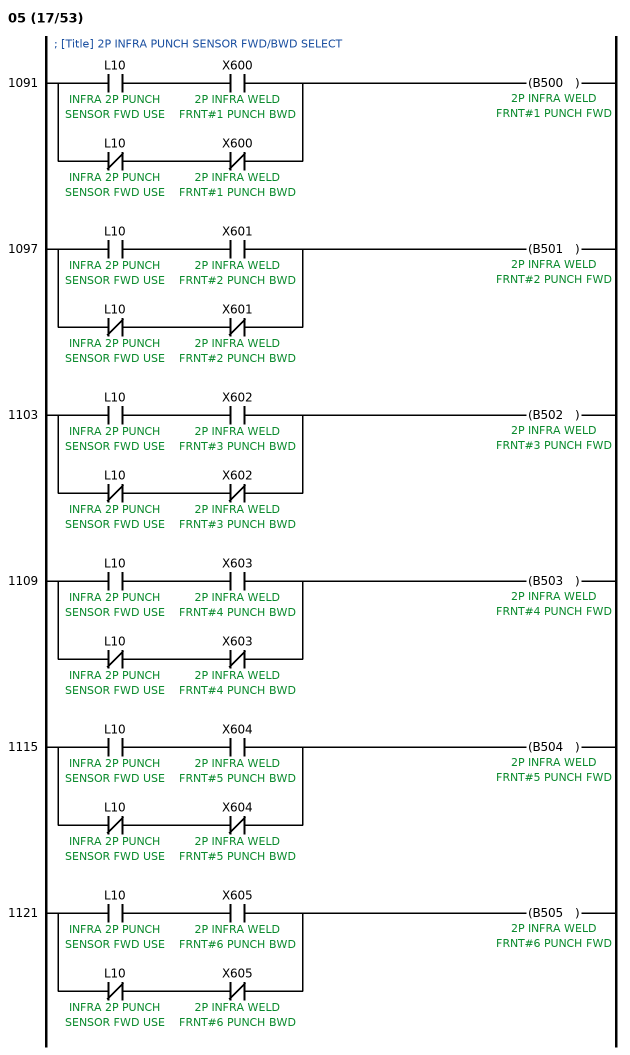
; [Title] 2P INFRA PUNCH SENSOR FWD/BWD SELECT
1091  LD      L10  ; INFRA 2P PUNCH SENSOR FWD USE
      AND     X600  ; 2P INFRA WELD FRNT#1 PUNCH BWD
      LDI     L10  ; INFRA 2P PUNCH SENSOR FWD USE
      ANI     X600  ; 2P INFRA WELD FRNT#1 PUNCH BWD
      ORB
      OUT     B500  ; 2P INFRA WELD FRNT#1 PUNCH FWD
1097  LD      L10  ; INFRA 2P PUNCH SENSOR FWD USE
      AND     X601  ; 2P INFRA WELD FRNT#2 PUNCH BWD
      LDI     L10  ; INFRA 2P PUNCH SENSOR FWD USE
      ANI     X601  ; 2P INFRA WELD FRNT#2 PUNCH BWD
      ORB
      OUT     B501  ; 2P INFRA WELD FRNT#2 PUNCH FWD
1103  LD      L10  ; INFRA 2P PUNCH SENSOR FWD USE
      AND     X602  ; 2P INFRA WELD FRNT#3 PUNCH BWD
      LDI     L10  ; INFRA 2P PUNCH SENSOR FWD USE
      ANI     X602  ; 2P INFRA WELD FRNT#3 PUNCH BWD
      ORB
      OUT     B502  ; 2P INFRA WELD FRNT#3 PUNCH FWD
1109  LD      L10  ; INFRA 2P PUNCH SENSOR FWD USE
      AND     X603  ; 2P INFRA WELD FRNT#4 PUNCH BWD
      LDI     L10  ; INFRA 2P PUNCH SENSOR FWD USE
      ANI     X603  ; 2P INFRA WELD FRNT#4 PUNCH BWD
      ORB
      OUT     B503  ; 2P INFRA WELD FRNT#4 PUNCH FWD
1115  LD      L10  ; INFRA 2P PUNCH SENSOR FWD USE
      AND     X604  ; 2P INFRA WELD FRNT#5 PUNCH BWD
      LDI     L10  ; INFRA 2P PUNCH SENSOR FWD USE
      ANI     X604  ; 2P INFRA WELD FRNT#5 PUNCH BWD
      ORB
      OUT     B504  ; 2P INFRA WELD FRNT#5 PUNCH FWD
1121  LD      L10  ; INFRA 2P PUNCH SENSOR FWD USE
      AND     X605  ; 2P INFRA WELD FRNT#6 PUNCH BWD
      LDI     L10  ; INFRA 2P PUNCH SENSOR FWD USE
      ANI     X605  ; 2P INFRA WELD FRNT#6 PUNCH BWD
      ORB
      OUT     B505  ; 2P INFRA WELD FRNT#6 PUNCH FWD
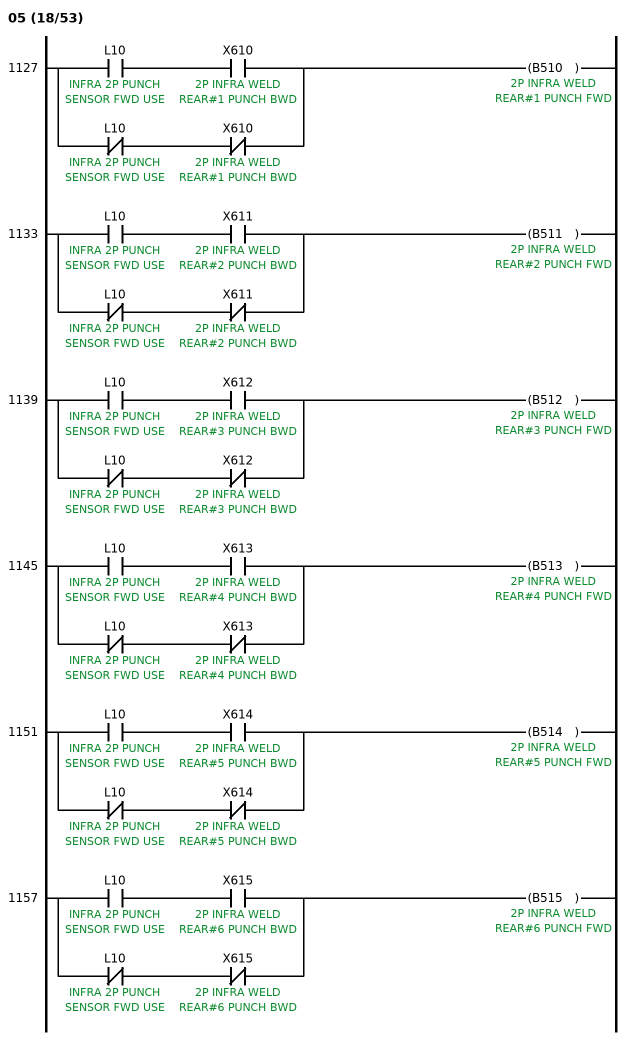
1127  LD      L10  ; INFRA 2P PUNCH SENSOR FWD USE
      AND     X610  ; 2P INFRA WELD REAR#1 PUNCH BWD
      LDI     L10  ; INFRA 2P PUNCH SENSOR FWD USE
      ANI     X610  ; 2P INFRA WELD REAR#1 PUNCH BWD
      ORB
      OUT     B510  ; 2P INFRA WELD REAR#1 PUNCH FWD
1133  LD      L10  ; INFRA 2P PUNCH SENSOR FWD USE
      AND     X611  ; 2P INFRA WELD REAR#2 PUNCH BWD
      LDI     L10  ; INFRA 2P PUNCH SENSOR FWD USE
      ANI     X611  ; 2P INFRA WELD REAR#2 PUNCH BWD
      ORB
      OUT     B511  ; 2P INFRA WELD REAR#2 PUNCH FWD
1139  LD      L10  ; INFRA 2P PUNCH SENSOR FWD USE
      AND     X612  ; 2P INFRA WELD REAR#3 PUNCH BWD
      LDI     L10  ; INFRA 2P PUNCH SENSOR FWD USE
      ANI     X612  ; 2P INFRA WELD REAR#3 PUNCH BWD
      ORB
      OUT     B512  ; 2P INFRA WELD REAR#3 PUNCH FWD
1145  LD      L10  ; INFRA 2P PUNCH SENSOR FWD USE
      AND     X613  ; 2P INFRA WELD REAR#4 PUNCH BWD
      LDI     L10  ; INFRA 2P PUNCH SENSOR FWD USE
      ANI     X613  ; 2P INFRA WELD REAR#4 PUNCH BWD
      ORB
      OUT     B513  ; 2P INFRA WELD REAR#4 PUNCH FWD
1151  LD      L10  ; INFRA 2P PUNCH SENSOR FWD USE
      AND     X614  ; 2P INFRA WELD REAR#5 PUNCH BWD
      LDI     L10  ; INFRA 2P PUNCH SENSOR FWD USE
      ANI     X614  ; 2P INFRA WELD REAR#5 PUNCH BWD
      ORB
      OUT     B514  ; 2P INFRA WELD REAR#5 PUNCH FWD
1157  LD      L10  ; INFRA 2P PUNCH SENSOR FWD USE
      AND     X615  ; 2P INFRA WELD REAR#6 PUNCH BWD
      LDI     L10  ; INFRA 2P PUNCH SENSOR FWD USE
      ANI     X615  ; 2P INFRA WELD REAR#6 PUNCH BWD
      ORB
      OUT     B515  ; 2P INFRA WELD REAR#6 PUNCH FWD
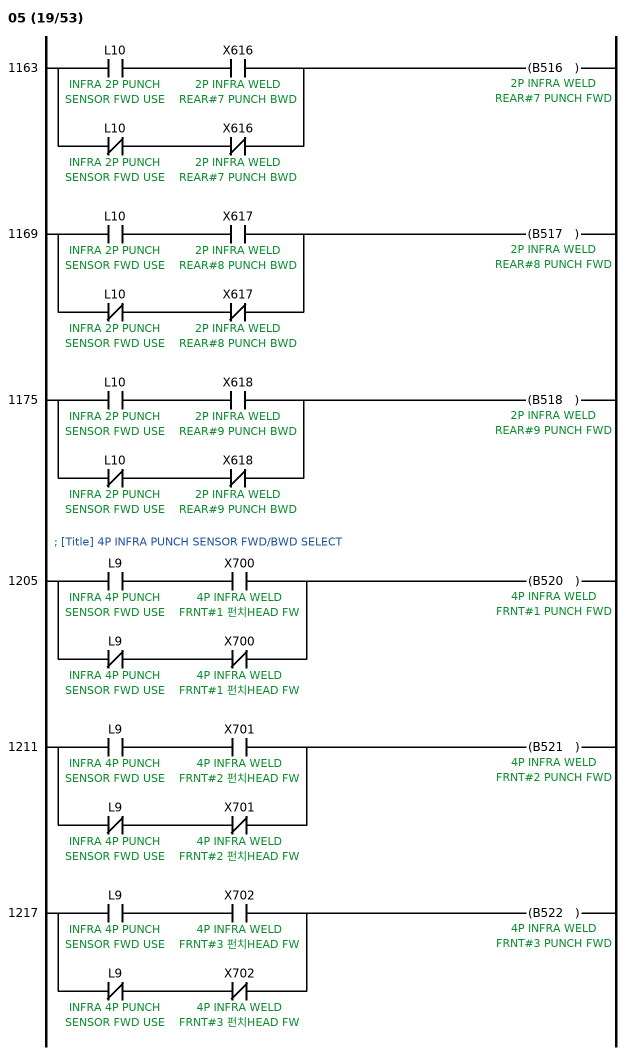
1163  LD      L10  ; INFRA 2P PUNCH SENSOR FWD USE
      AND     X616  ; 2P INFRA WELD REAR#7 PUNCH BWD
      LDI     L10  ; INFRA 2P PUNCH SENSOR FWD USE
      ANI     X616  ; 2P INFRA WELD REAR#7 PUNCH BWD
      ORB
      OUT     B516  ; 2P INFRA WELD REAR#7 PUNCH FWD
1169  LD      L10  ; INFRA 2P PUNCH SENSOR FWD USE
      AND     X617  ; 2P INFRA WELD REAR#8 PUNCH BWD
      LDI     L10  ; INFRA 2P PUNCH SENSOR FWD USE
      ANI     X617  ; 2P INFRA WELD REAR#8 PUNCH BWD
      ORB
      OUT     B517  ; 2P INFRA WELD REAR#8 PUNCH FWD
1175  LD      L10  ; INFRA 2P PUNCH SENSOR FWD USE
      AND     X618  ; 2P INFRA WELD REAR#9 PUNCH BWD
      LDI     L10  ; INFRA 2P PUNCH SENSOR FWD USE
      ANI     X618  ; 2P INFRA WELD REAR#9 PUNCH BWD
      ORB
      OUT     B518  ; 2P INFRA WELD REAR#9 PUNCH FWD
; [Title] 4P INFRA PUNCH SENSOR FWD/BWD SELECT
1205  LD      L9  ; INFRA 4P PUNCH SENSOR FWD USE
      AND     X700  ; 4P INFRA WELD FRNT#1 펀치HEAD FW
      LDI     L9  ; INFRA 4P PUNCH SENSOR FWD USE
      ANI     X700  ; 4P INFRA WELD FRNT#1 펀치HEAD FW
      ORB
      OUT     B520  ; 4P INFRA WELD FRNT#1 PUNCH FWD
1211  LD      L9  ; INFRA 4P PUNCH SENSOR FWD USE
      AND     X701  ; 4P INFRA WELD FRNT#2 펀치HEAD FW
      LDI     L9  ; INFRA 4P PUNCH SENSOR FWD USE
      ANI     X701  ; 4P INFRA WELD FRNT#2 펀치HEAD FW
      ORB
      OUT     B521  ; 4P INFRA WELD FRNT#2 PUNCH FWD
1217  LD      L9  ; INFRA 4P PUNCH SENSOR FWD USE
      AND     X702  ; 4P INFRA WELD FRNT#3 펀치HEAD FW
      LDI     L9  ; INFRA 4P PUNCH SENSOR FWD USE
      ANI     X702  ; 4P INFRA WELD FRNT#3 펀치HEAD FW
      ORB
      OUT     B522  ; 4P INFRA WELD FRNT#3 PUNCH FWD
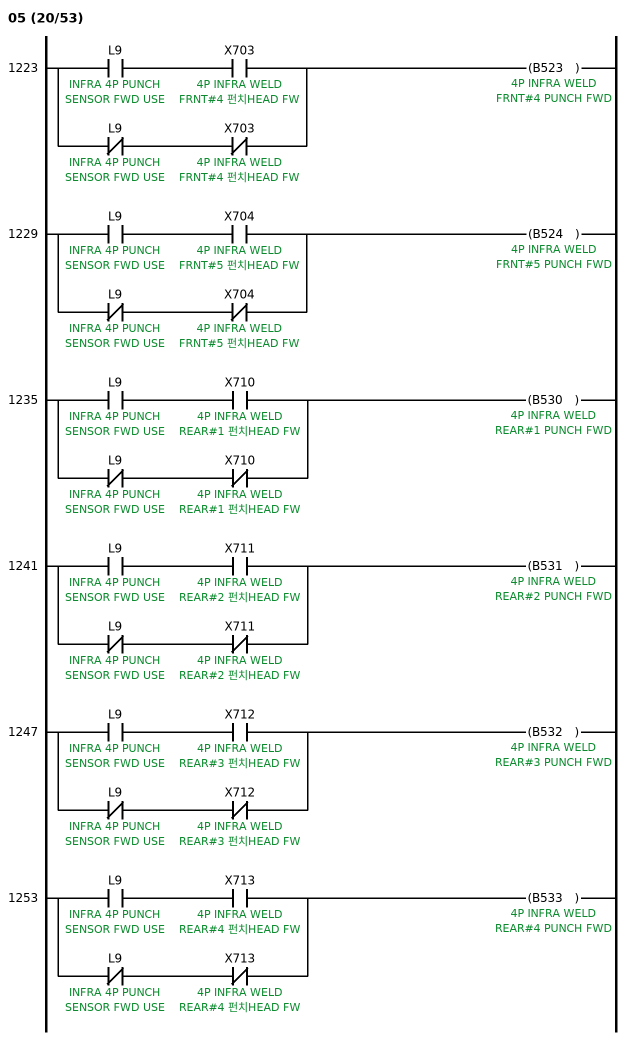
1223  LD      L9  ; INFRA 4P PUNCH SENSOR FWD USE
      AND     X703  ; 4P INFRA WELD FRNT#4 펀치HEAD FW
      LDI     L9  ; INFRA 4P PUNCH SENSOR FWD USE
      ANI     X703  ; 4P INFRA WELD FRNT#4 펀치HEAD FW
      ORB
      OUT     B523  ; 4P INFRA WELD FRNT#4 PUNCH FWD
1229  LD      L9  ; INFRA 4P PUNCH SENSOR FWD USE
      AND     X704  ; 4P INFRA WELD FRNT#5 펀치HEAD FW
      LDI     L9  ; INFRA 4P PUNCH SENSOR FWD USE
      ANI     X704  ; 4P INFRA WELD FRNT#5 펀치HEAD FW
      ORB
      OUT     B524  ; 4P INFRA WELD FRNT#5 PUNCH FWD
1235  LD      L9  ; INFRA 4P PUNCH SENSOR FWD USE
      AND     X710  ; 4P INFRA WELD REAR#1 펀치HEAD FW
      LDI     L9  ; INFRA 4P PUNCH SENSOR FWD USE
      ANI     X710  ; 4P INFRA WELD REAR#1 펀치HEAD FW
      ORB
      OUT     B530  ; 4P INFRA WELD REAR#1 PUNCH FWD
1241  LD      L9  ; INFRA 4P PUNCH SENSOR FWD USE
      AND     X711  ; 4P INFRA WELD REAR#2 펀치HEAD FW
      LDI     L9  ; INFRA 4P PUNCH SENSOR FWD USE
      ANI     X711  ; 4P INFRA WELD REAR#2 펀치HEAD FW
      ORB
      OUT     B531  ; 4P INFRA WELD REAR#2 PUNCH FWD
1247  LD      L9  ; INFRA 4P PUNCH SENSOR FWD USE
      AND     X712  ; 4P INFRA WELD REAR#3 펀치HEAD FW
      LDI     L9  ; INFRA 4P PUNCH SENSOR FWD USE
      ANI     X712  ; 4P INFRA WELD REAR#3 펀치HEAD FW
      ORB
      OUT     B532  ; 4P INFRA WELD REAR#3 PUNCH FWD
1253  LD      L9  ; INFRA 4P PUNCH SENSOR FWD USE
      AND     X713  ; 4P INFRA WELD REAR#4 펀치HEAD FW
      LDI     L9  ; INFRA 4P PUNCH SENSOR FWD USE
      ANI     X713  ; 4P INFRA WELD REAR#4 펀치HEAD FW
      ORB
      OUT     B533  ; 4P INFRA WELD REAR#4 PUNCH FWD
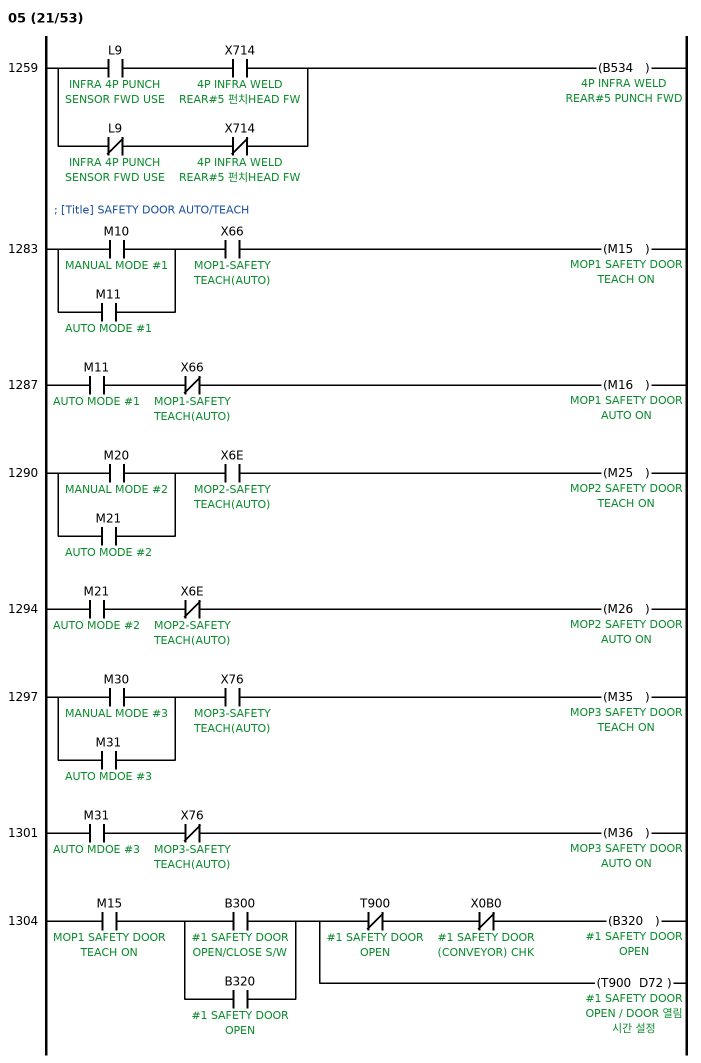
1259  LD      L9  ; INFRA 4P PUNCH SENSOR FWD USE
      AND     X714  ; 4P INFRA WELD REAR#5 펀치HEAD FW
      LDI     L9  ; INFRA 4P PUNCH SENSOR FWD USE
      ANI     X714  ; 4P INFRA WELD REAR#5 펀치HEAD FW
      ORB
      OUT     B534  ; 4P INFRA WELD REAR#5 PUNCH FWD
; [Title] SAFETY DOOR AUTO/TEACH
1283  LD      M10  ; MANUAL MODE #1
      OR      M11  ; AUTO MODE #1
      AND     X66  ; MOP1-SAFETY TEACH(AUTO)
      OUT     M15  ; MOP1 SAFETY DOOR TEACH ON
1287  LD      M11  ; AUTO MODE #1
      ANI     X66  ; MOP1-SAFETY TEACH(AUTO)
      OUT     M16  ; MOP1 SAFETY DOOR AUTO ON
1290  LD      M20  ; MANUAL MODE #2
      OR      M21  ; AUTO MODE #2
      AND     X6E  ; MOP2-SAFETY TEACH(AUTO)
      OUT     M25  ; MOP2 SAFETY DOOR TEACH ON
1294  LD      M21  ; AUTO MODE #2
      ANI     X6E  ; MOP2-SAFETY TEACH(AUTO)
      OUT     M26  ; MOP2 SAFETY DOOR AUTO ON
1297  LD      M30  ; MANUAL MODE #3
      OR      M31  ; AUTO MDOE #3
      AND     X76  ; MOP3-SAFETY TEACH(AUTO)
      OUT     M35  ; MOP3 SAFETY DOOR TEACH ON
1301  LD      M31  ; AUTO MDOE #3
      ANI     X76  ; MOP3-SAFETY TEACH(AUTO)
      OUT     M36  ; MOP3 SAFETY DOOR AUTO ON
1304  LD      M15  ; MOP1 SAFETY DOOR TEACH ON
      LD      B300  ; #1 SAFETY DOOR  OPEN/CLOSE S/W
      OR      B320  ; #1 SAFETY DOOR  OPEN
      ANB
      MPS
      ANI     T900  ; #1 SAFETY DOOR  OPEN
      ANI     X0B0  ; #1 SAFETY DOOR (CONVEYOR) CHK
      OUT     B320  ; #1 SAFETY DOOR  OPEN
      MPP
      OUT     T900 D72  ; #1 SAFETY DOOR  OPEN / DOOR 열림 시간 설정
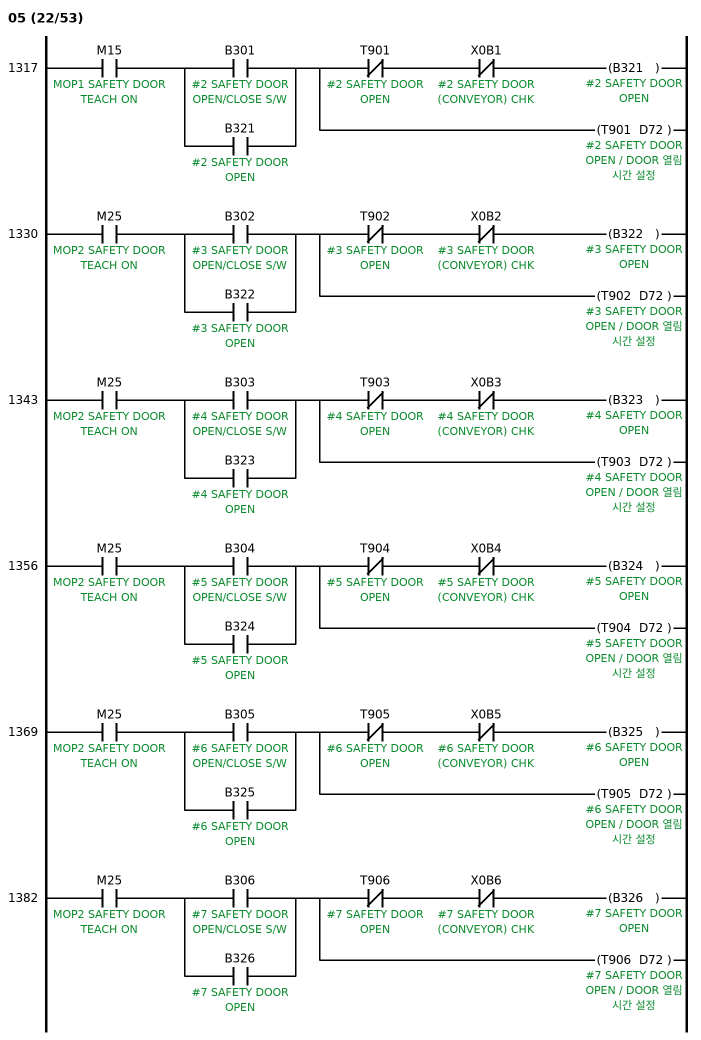
1317  LD      M15  ; MOP1 SAFETY DOOR TEACH ON
      LD      B301  ; #2 SAFETY DOOR  OPEN/CLOSE S/W
      OR      B321  ; #2 SAFETY DOOR  OPEN
      ANB
      MPS
      ANI     T901  ; #2 SAFETY DOOR  OPEN
      ANI     X0B1  ; #2 SAFETY DOOR (CONVEYOR) CHK
      OUT     B321  ; #2 SAFETY DOOR  OPEN
      MPP
      OUT     T901 D72  ; #2 SAFETY DOOR  OPEN / DOOR 열림 시간 설정
1330  LD      M25  ; MOP2 SAFETY DOOR TEACH ON
      LD      B302  ; #3 SAFETY DOOR  OPEN/CLOSE S/W
      OR      B322  ; #3 SAFETY DOOR  OPEN
      ANB
      MPS
      ANI     T902  ; #3 SAFETY DOOR  OPEN
      ANI     X0B2  ; #3 SAFETY DOOR (CONVEYOR) CHK
      OUT     B322  ; #3 SAFETY DOOR  OPEN
      MPP
      OUT     T902 D72  ; #3 SAFETY DOOR  OPEN / DOOR 열림 시간 설정
1343  LD      M25  ; MOP2 SAFETY DOOR TEACH ON
      LD      B303  ; #4 SAFETY DOOR  OPEN/CLOSE S/W
      OR      B323  ; #4 SAFETY DOOR  OPEN
      ANB
      MPS
      ANI     T903  ; #4 SAFETY DOOR  OPEN
      ANI     X0B3  ; #4 SAFETY DOOR (CONVEYOR) CHK
      OUT     B323  ; #4 SAFETY DOOR  OPEN
      MPP
      OUT     T903 D72  ; #4 SAFETY DOOR  OPEN / DOOR 열림 시간 설정
1356  LD      M25  ; MOP2 SAFETY DOOR TEACH ON
      LD      B304  ; #5 SAFETY DOOR  OPEN/CLOSE S/W
      OR      B324  ; #5 SAFETY DOOR  OPEN
      ANB
      MPS
      ANI     T904  ; #5 SAFETY DOOR  OPEN
      ANI     X0B4  ; #5 SAFETY DOOR (CONVEYOR) CHK
      OUT     B324  ; #5 SAFETY DOOR  OPEN
      MPP
      OUT     T904 D72  ; #5 SAFETY DOOR  OPEN / DOOR 열림 시간 설정
1369  LD      M25  ; MOP2 SAFETY DOOR TEACH ON
      LD      B305  ; #6 SAFETY DOOR  OPEN/CLOSE S/W
      OR      B325  ; #6 SAFETY DOOR  OPEN
      ANB
      MPS
      ANI     T905  ; #6 SAFETY DOOR  OPEN
      ANI     X0B5  ; #6 SAFETY DOOR (CONVEYOR) CHK
      OUT     B325  ; #6 SAFETY DOOR  OPEN
      MPP
      OUT     T905 D72  ; #6 SAFETY DOOR  OPEN / DOOR 열림 시간 설정
1382  LD      M25  ; MOP2 SAFETY DOOR TEACH ON
      LD      B306  ; #7 SAFETY DOOR  OPEN/CLOSE S/W
      OR      B326  ; #7 SAFETY DOOR  OPEN
      ANB
      MPS
      ANI     T906  ; #7 SAFETY DOOR  OPEN
      ANI     X0B6  ; #7 SAFETY DOOR (CONVEYOR) CHK
      OUT     B326  ; #7 SAFETY DOOR  OPEN
      MPP
      OUT     T906 D72  ; #7 SAFETY DOOR  OPEN / DOOR 열림 시간 설정
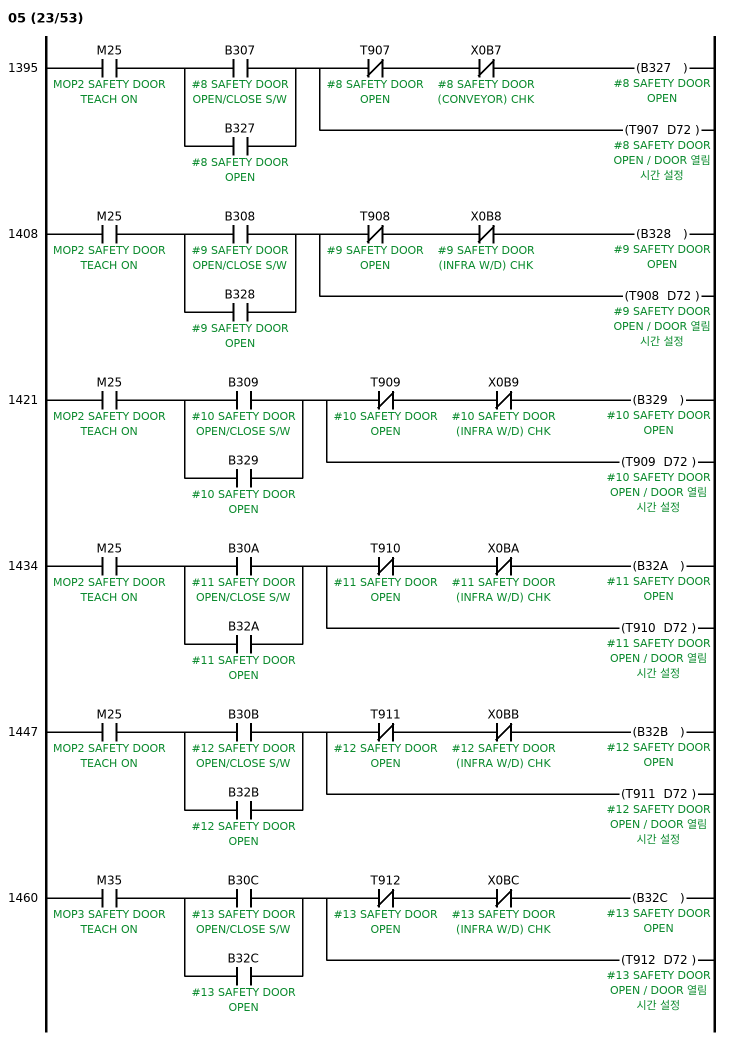
1395  LD      M25  ; MOP2 SAFETY DOOR TEACH ON
      LD      B307  ; #8 SAFETY DOOR  OPEN/CLOSE S/W
      OR      B327  ; #8 SAFETY DOOR  OPEN
      ANB
      MPS
      ANI     T907  ; #8 SAFETY DOOR  OPEN
      ANI     X0B7  ; #8 SAFETY DOOR (CONVEYOR) CHK
      OUT     B327  ; #8 SAFETY DOOR  OPEN
      MPP
      OUT     T907 D72  ; #8 SAFETY DOOR  OPEN / DOOR 열림 시간 설정
1408  LD      M25  ; MOP2 SAFETY DOOR TEACH ON
      LD      B308  ; #9 SAFETY DOOR  OPEN/CLOSE S/W
      OR      B328  ; #9 SAFETY DOOR  OPEN
      ANB
      MPS
      ANI     T908  ; #9 SAFETY DOOR  OPEN
      ANI     X0B8  ; #9 SAFETY DOOR (INFRA W/D) CHK
      OUT     B328  ; #9 SAFETY DOOR  OPEN
      MPP
      OUT     T908 D72  ; #9 SAFETY DOOR  OPEN / DOOR 열림 시간 설정
1421  LD      M25  ; MOP2 SAFETY DOOR TEACH ON
      LD      B309  ; #10 SAFETY DOOR OPEN/CLOSE S/W
      OR      B329  ; #10 SAFETY DOOR OPEN
      ANB
      MPS
      ANI     T909  ; #10 SAFETY DOOR OPEN
      ANI     X0B9  ; #10 SAFETY DOOR (INFRA W/D) CHK
      OUT     B329  ; #10 SAFETY DOOR OPEN
      MPP
      OUT     T909 D72  ; #10 SAFETY DOOR OPEN / DOOR 열림 시간 설정
1434  LD      M25  ; MOP2 SAFETY DOOR TEACH ON
      LD      B30A  ; #11 SAFETY DOOR OPEN/CLOSE S/W
      OR      B32A  ; #11 SAFETY DOOR OPEN
      ANB
      MPS
      ANI     T910  ; #11 SAFETY DOOR OPEN
      ANI     X0BA  ; #11 SAFETY DOOR (INFRA W/D) CHK
      OUT     B32A  ; #11 SAFETY DOOR OPEN
      MPP
      OUT     T910 D72  ; #11 SAFETY DOOR OPEN / DOOR 열림 시간 설정
1447  LD      M25  ; MOP2 SAFETY DOOR TEACH ON
      LD      B30B  ; #12 SAFETY DOOR OPEN/CLOSE S/W
      OR      B32B  ; #12 SAFETY DOOR OPEN
      ANB
      MPS
      ANI     T911  ; #12 SAFETY DOOR OPEN
      ANI     X0BB  ; #12 SAFETY DOOR (INFRA W/D) CHK
      OUT     B32B  ; #12 SAFETY DOOR OPEN
      MPP
      OUT     T911 D72  ; #12 SAFETY DOOR OPEN / DOOR 열림 시간 설정
1460  LD      M35  ; MOP3 SAFETY DOOR TEACH ON
      LD      B30C  ; #13 SAFETY DOOR OPEN/CLOSE S/W
      OR      B32C  ; #13 SAFETY DOOR OPEN
      ANB
      MPS
      ANI     T912  ; #13 SAFETY DOOR OPEN
      ANI     X0BC  ; #13 SAFETY DOOR (INFRA W/D) CHK
      OUT     B32C  ; #13 SAFETY DOOR OPEN
      MPP
      OUT     T912 D72  ; #13 SAFETY DOOR OPEN / DOOR 열림 시간 설정
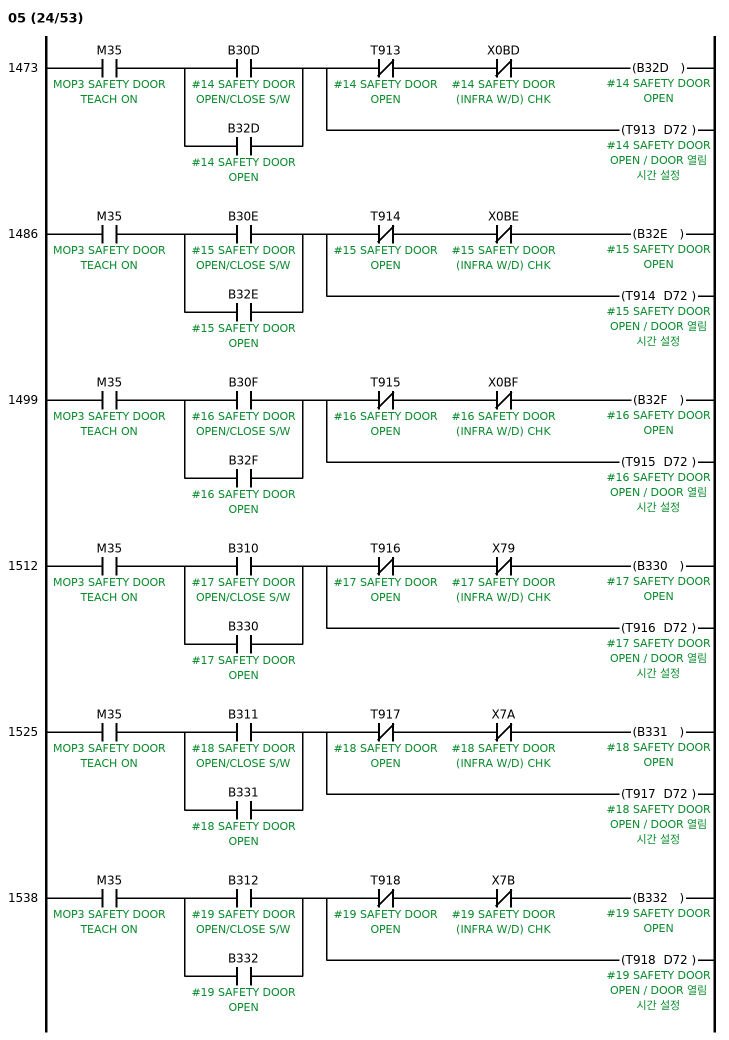
1473  LD      M35  ; MOP3 SAFETY DOOR TEACH ON
      LD      B30D  ; #14 SAFETY DOOR OPEN/CLOSE S/W
      OR      B32D  ; #14 SAFETY DOOR OPEN
      ANB
      MPS
      ANI     T913  ; #14 SAFETY DOOR OPEN
      ANI     X0BD  ; #14 SAFETY DOOR (INFRA W/D) CHK
      OUT     B32D  ; #14 SAFETY DOOR OPEN
      MPP
      OUT     T913 D72  ; #14 SAFETY DOOR OPEN / DOOR 열림 시간 설정
1486  LD      M35  ; MOP3 SAFETY DOOR TEACH ON
      LD      B30E  ; #15 SAFETY DOOR OPEN/CLOSE S/W
      OR      B32E  ; #15 SAFETY DOOR OPEN
      ANB
      MPS
      ANI     T914  ; #15 SAFETY DOOR OPEN
      ANI     X0BE  ; #15 SAFETY DOOR (INFRA W/D) CHK
      OUT     B32E  ; #15 SAFETY DOOR OPEN
      MPP
      OUT     T914 D72  ; #15 SAFETY DOOR OPEN / DOOR 열림 시간 설정
1499  LD      M35  ; MOP3 SAFETY DOOR TEACH ON
      LD      B30F  ; #16 SAFETY DOOR OPEN/CLOSE S/W
      OR      B32F  ; #16 SAFETY DOOR OPEN
      ANB
      MPS
      ANI     T915  ; #16 SAFETY DOOR OPEN
      ANI     X0BF  ; #16 SAFETY DOOR (INFRA W/D) CHK
      OUT     B32F  ; #16 SAFETY DOOR OPEN
      MPP
      OUT     T915 D72  ; #16 SAFETY DOOR OPEN / DOOR 열림 시간 설정
1512  LD      M35  ; MOP3 SAFETY DOOR TEACH ON
      LD      B310  ; #17 SAFETY DOOR OPEN/CLOSE S/W
      OR      B330  ; #17 SAFETY DOOR OPEN
      ANB
      MPS
      ANI     T916  ; #17 SAFETY DOOR OPEN
      ANI     X79  ; #17 SAFETY DOOR (INFRA W/D) CHK
      OUT     B330  ; #17 SAFETY DOOR OPEN
      MPP
      OUT     T916 D72  ; #17 SAFETY DOOR OPEN / DOOR 열림 시간 설정
1525  LD      M35  ; MOP3 SAFETY DOOR TEACH ON
      LD      B311  ; #18 SAFETY DOOR OPEN/CLOSE S/W
      OR      B331  ; #18 SAFETY DOOR OPEN
      ANB
      MPS
      ANI     T917  ; #18 SAFETY DOOR OPEN
      ANI     X7A  ; #18 SAFETY DOOR (INFRA W/D) CHK
      OUT     B331  ; #18 SAFETY DOOR OPEN
      MPP
      OUT     T917 D72  ; #18 SAFETY DOOR OPEN / DOOR 열림 시간 설정
1538  LD      M35  ; MOP3 SAFETY DOOR TEACH ON
      LD      B312  ; #19 SAFETY DOOR OPEN/CLOSE S/W
      OR      B332  ; #19 SAFETY DOOR OPEN
      ANB
      MPS
      ANI     T918  ; #19 SAFETY DOOR OPEN
      ANI     X7B  ; #19 SAFETY DOOR (INFRA W/D) CHK
      OUT     B332  ; #19 SAFETY DOOR OPEN
      MPP
      OUT     T918 D72  ; #19 SAFETY DOOR OPEN / DOOR 열림 시간 설정
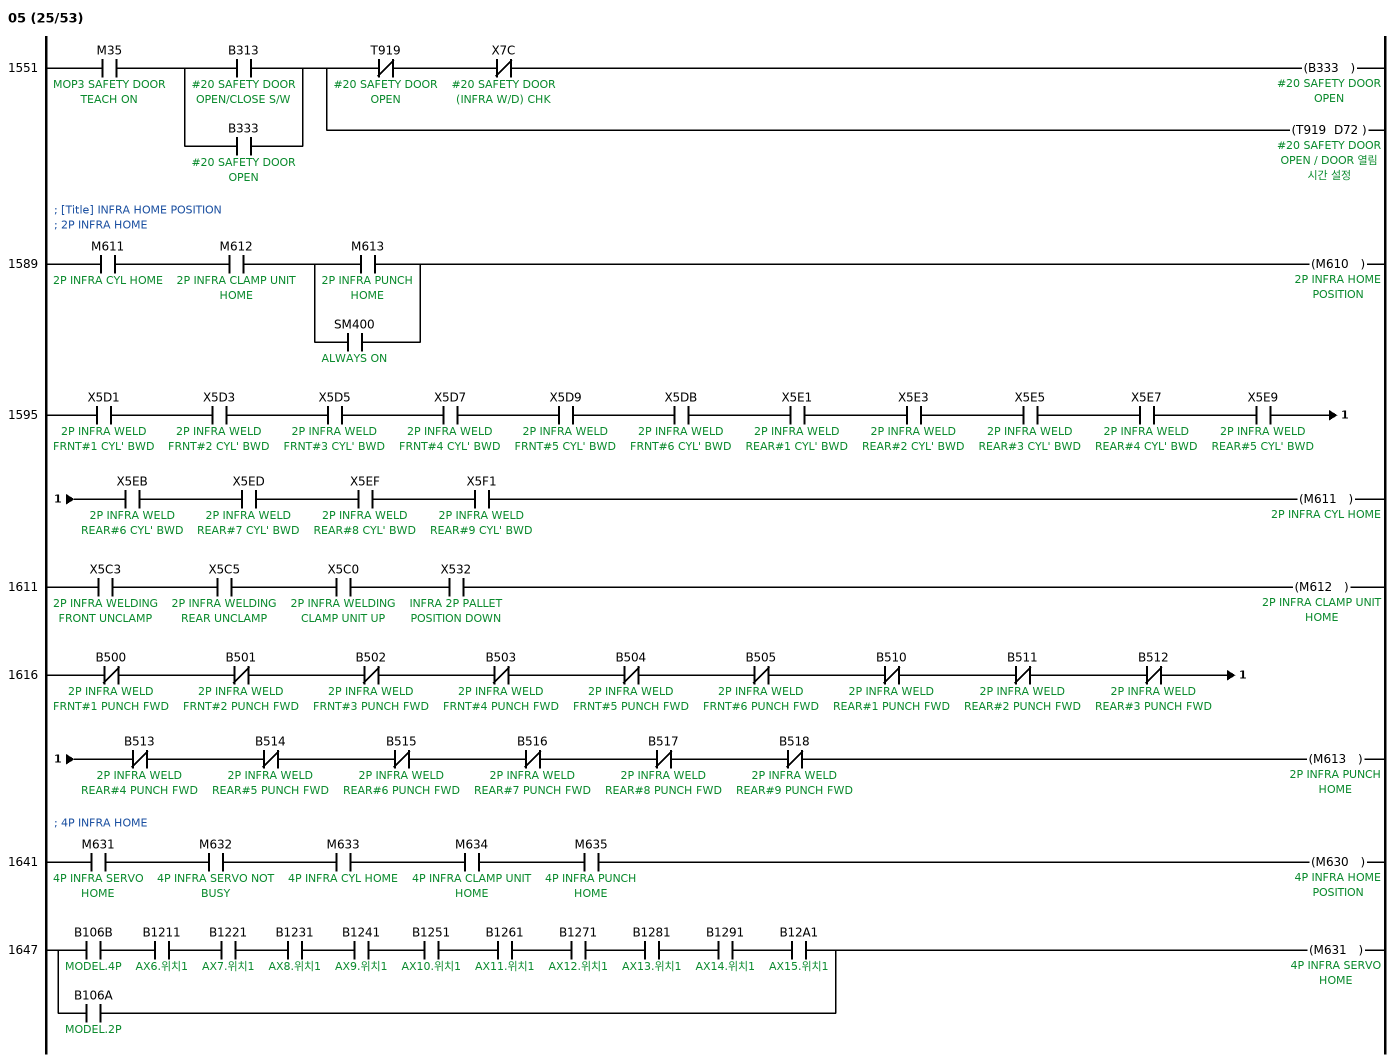
1551  LD      M35  ; MOP3 SAFETY DOOR TEACH ON
      LD      B313  ; #20 SAFETY DOOR OPEN/CLOSE S/W
      OR      B333  ; #20 SAFETY DOOR OPEN
      ANB
      MPS
      ANI     T919  ; #20 SAFETY DOOR OPEN
      ANI     X7C  ; #20 SAFETY DOOR (INFRA W/D) CHK
      OUT     B333  ; #20 SAFETY DOOR OPEN
      MPP
      OUT     T919 D72  ; #20 SAFETY DOOR OPEN / DOOR 열림 시간 설정
; [Title] INFRA HOME POSITION
; 2P INFRA HOME
1589  LD      M611  ; 2P INFRA CYL HOME
      AND     M612  ; 2P INFRA CLAMP UNIT HOME
      LD      M613  ; 2P INFRA PUNCH HOME
      OR      SM400  ; ALWAYS ON
      ANB
      OUT     M610  ; 2P INFRA HOME POSITION
1595  LD      X5D1  ; 2P INFRA WELD FRNT#1 CYL' BWD
      AND     X5D3  ; 2P INFRA WELD FRNT#2 CYL' BWD
      AND     X5D5  ; 2P INFRA WELD FRNT#3 CYL' BWD
      AND     X5D7  ; 2P INFRA WELD FRNT#4 CYL' BWD
      AND     X5D9  ; 2P INFRA WELD FRNT#5 CYL' BWD
      AND     X5DB  ; 2P INFRA WELD FRNT#6 CYL' BWD
      AND     X5E1  ; 2P INFRA WELD REAR#1 CYL' BWD
      AND     X5E3  ; 2P INFRA WELD REAR#2 CYL' BWD
      AND     X5E5  ; 2P INFRA WELD REAR#3 CYL' BWD
      AND     X5E7  ; 2P INFRA WELD REAR#4 CYL' BWD
      AND     X5E9  ; 2P INFRA WELD REAR#5 CYL' BWD
      AND     X5EB  ; 2P INFRA WELD REAR#6 CYL' BWD
      AND     X5ED  ; 2P INFRA WELD REAR#7 CYL' BWD
      AND     X5EF  ; 2P INFRA WELD REAR#8 CYL' BWD
      AND     X5F1  ; 2P INFRA WELD REAR#9 CYL' BWD
      OUT     M611  ; 2P INFRA CYL HOME
1611  LD      X5C3  ; 2P INFRA WELDING FRONT UNCLAMP
      AND     X5C5  ; 2P INFRA WELDING REAR UNCLAMP
      AND     X5C0  ; 2P INFRA WELDING CLAMP UNIT UP
      AND     X532  ; INFRA 2P PALLET POSITION DOWN
      OUT     M612  ; 2P INFRA CLAMP UNIT HOME
1616  LDI     B500  ; 2P INFRA WELD FRNT#1 PUNCH FWD
      ANI     B501  ; 2P INFRA WELD FRNT#2 PUNCH FWD
      ANI     B502  ; 2P INFRA WELD FRNT#3 PUNCH FWD
      ANI     B503  ; 2P INFRA WELD FRNT#4 PUNCH FWD
      ANI     B504  ; 2P INFRA WELD FRNT#5 PUNCH FWD
      ANI     B505  ; 2P INFRA WELD FRNT#6 PUNCH FWD
      ANI     B510  ; 2P INFRA WELD REAR#1 PUNCH FWD
      ANI     B511  ; 2P INFRA WELD REAR#2 PUNCH FWD
      ANI     B512  ; 2P INFRA WELD REAR#3 PUNCH FWD
      ANI     B513  ; 2P INFRA WELD REAR#4 PUNCH FWD
      ANI     B514  ; 2P INFRA WELD REAR#5 PUNCH FWD
      ANI     B515  ; 2P INFRA WELD REAR#6 PUNCH FWD
      ANI     B516  ; 2P INFRA WELD REAR#7 PUNCH FWD
      ANI     B517  ; 2P INFRA WELD REAR#8 PUNCH FWD
      ANI     B518  ; 2P INFRA WELD REAR#9 PUNCH FWD
      OUT     M613  ; 2P INFRA PUNCH HOME
; 4P INFRA HOME
1641  LD      M631  ; 4P INFRA SERVO HOME
      AND     M632  ; 4P INFRA SERVO NOT BUSY
      AND     M633  ; 4P INFRA CYL HOME
      AND     M634  ; 4P INFRA CLAMP UNIT HOME
      AND     M635  ; 4P INFRA PUNCH HOME
      OUT     M630  ; 4P INFRA HOME POSITION
1647  LD      B106B  ; MODEL.4P
      AND     B1211  ; AX6.위치1
      AND     B1221  ; AX7.위치1
      AND     B1231  ; AX8.위치1
      AND     B1241  ; AX9.위치1
      AND     B1251  ; AX10.위치1
      AND     B1261  ; AX11.위치1
      AND     B1271  ; AX12.위치1
      AND     B1281  ; AX13.위치1
      AND     B1291  ; AX14.위치1
      AND     B12A1  ; AX15.위치1
      OR      B106A  ; MODEL.2P
      OUT     M631  ; 4P INFRA SERVO HOME
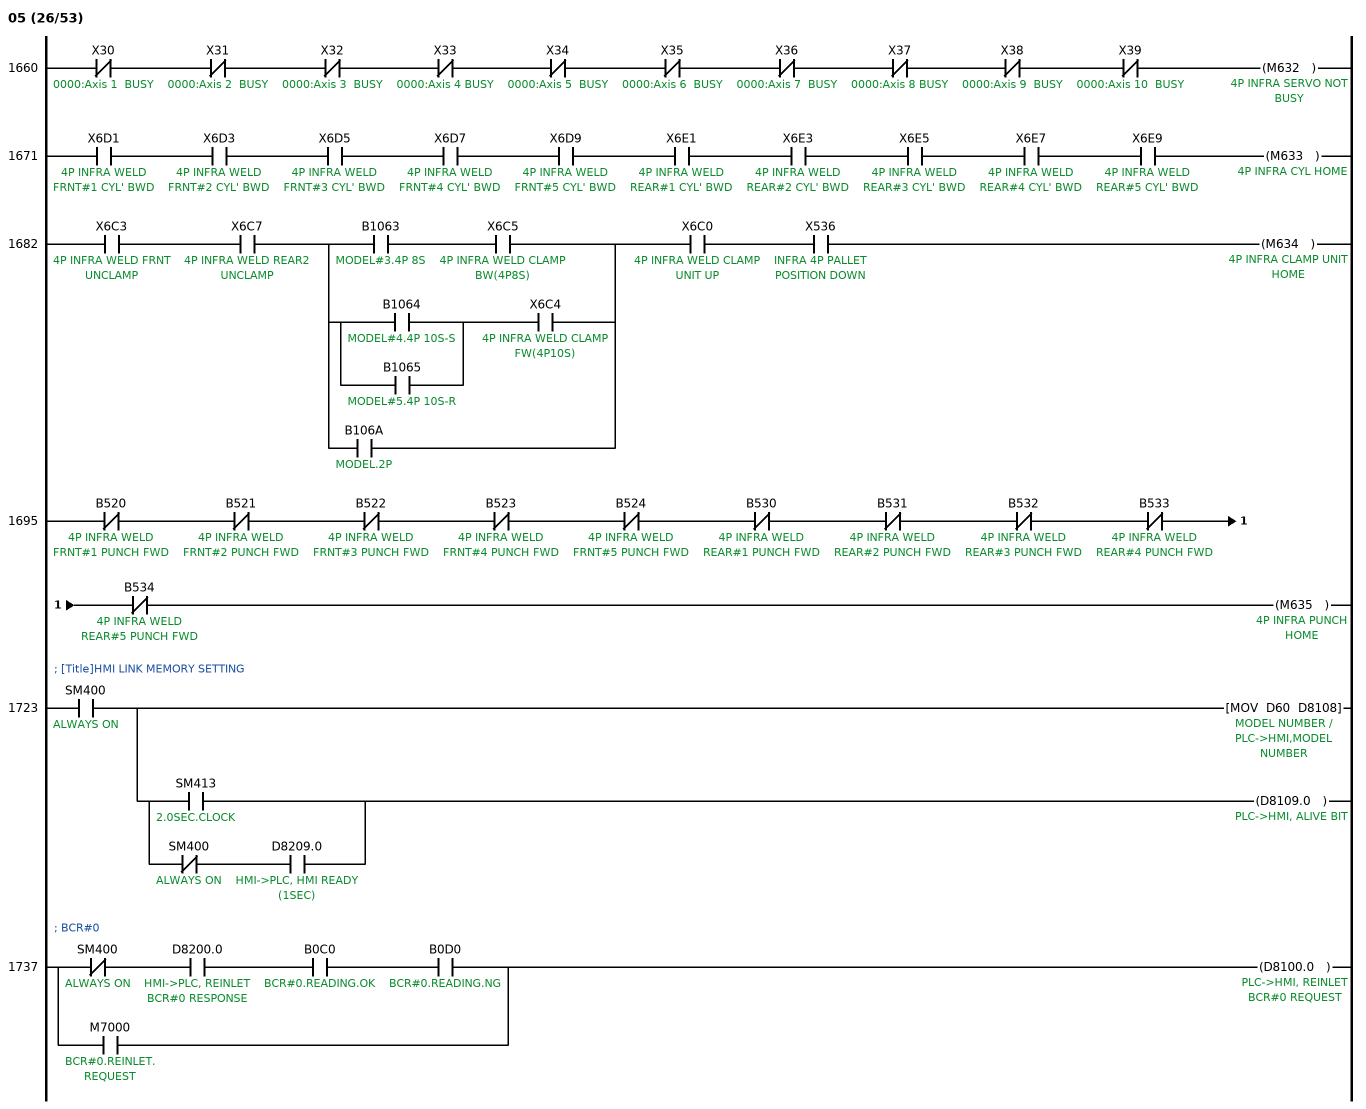
1660  LDI     X30  ; 0000:Axis 1  BUSY
      ANI     X31  ; 0000:Axis 2  BUSY
      ANI     X32  ; 0000:Axis 3  BUSY
      ANI     X33  ; 0000:Axis 4 BUSY
      ANI     X34  ; 0000:Axis 5  BUSY
      ANI     X35  ; 0000:Axis 6  BUSY
      ANI     X36  ; 0000:Axis 7  BUSY
      ANI     X37  ; 0000:Axis 8 BUSY
      ANI     X38  ; 0000:Axis 9  BUSY
      ANI     X39  ; 0000:Axis 10  BUSY
      OUT     M632  ; 4P INFRA SERVO NOT BUSY
1671  LD      X6D1  ; 4P INFRA WELD FRNT#1 CYL' BWD
      AND     X6D3  ; 4P INFRA WELD FRNT#2 CYL' BWD
      AND     X6D5  ; 4P INFRA WELD FRNT#3 CYL' BWD
      AND     X6D7  ; 4P INFRA WELD FRNT#4 CYL' BWD
      AND     X6D9  ; 4P INFRA WELD FRNT#5 CYL' BWD
      AND     X6E1  ; 4P INFRA WELD REAR#1 CYL' BWD
      AND     X6E3  ; 4P INFRA WELD REAR#2 CYL' BWD
      AND     X6E5  ; 4P INFRA WELD REAR#3 CYL' BWD
      AND     X6E7  ; 4P INFRA WELD REAR#4 CYL' BWD
      AND     X6E9  ; 4P INFRA WELD REAR#5 CYL' BWD
      OUT     M633  ; 4P INFRA CYL HOME
1682  LD      X6C3  ; 4P INFRA WELD FRNT UNCLAMP
      AND     X6C7  ; 4P INFRA WELD REAR2 UNCLAMP
      LD      B1063  ; MODEL#3.4P 8S
      AND     X6C5  ; 4P INFRA WELD CLAMP BW(4P8S)
      LD      B1064  ; MODEL#4.4P 10S-S
      OR      B1065  ; MODEL#5.4P 10S-R
      AND     X6C4  ; 4P INFRA WELD CLAMP FW(4P10S)
      ORB
      OR      B106A  ; MODEL.2P
      ANB
      AND     X6C0  ; 4P INFRA WELD CLAMP UNIT UP
      AND     X536  ; INFRA 4P PALLET POSITION DOWN
      OUT     M634  ; 4P INFRA CLAMP UNIT HOME
1695  LDI     B520  ; 4P INFRA WELD FRNT#1 PUNCH FWD
      ANI     B521  ; 4P INFRA WELD FRNT#2 PUNCH FWD
      ANI     B522  ; 4P INFRA WELD FRNT#3 PUNCH FWD
      ANI     B523  ; 4P INFRA WELD FRNT#4 PUNCH FWD
      ANI     B524  ; 4P INFRA WELD FRNT#5 PUNCH FWD
      ANI     B530  ; 4P INFRA WELD REAR#1 PUNCH FWD
      ANI     B531  ; 4P INFRA WELD REAR#2 PUNCH FWD
      ANI     B532  ; 4P INFRA WELD REAR#3 PUNCH FWD
      ANI     B533  ; 4P INFRA WELD REAR#4 PUNCH FWD
      ANI     B534  ; 4P INFRA WELD REAR#5 PUNCH FWD
      OUT     M635  ; 4P INFRA PUNCH HOME
; [Title]HMI LINK MEMORY SETTING
1723  LD      SM400  ; ALWAYS ON
      MOV     D60 D8108  ; PLC->HMI,MODEL NUMBER
      LD      SM413  ; 2.0SEC.CLOCK
      LDI     SM400  ; ALWAYS ON
      AND     D8209.0  ; HMI->PLC, HMI READY (1SEC)
      ORB
      ANB
      OUT     D8109.0  ; PLC->HMI, ALIVE BIT
; BCR#0
1737  LDI     SM400  ; ALWAYS ON
      AND     D8200.0  ; HMI->PLC, REINLET BCR#0 RESPONSE
      AND     B0C0  ; BCR#0.READING.OK
      AND     B0D0  ; BCR#0.READING.NG
      OR      M7000  ; BCR#0.REINLET.REQUEST
      OUT     D8100.0  ; PLC->HMI, REINLET BCR#0 REQUEST
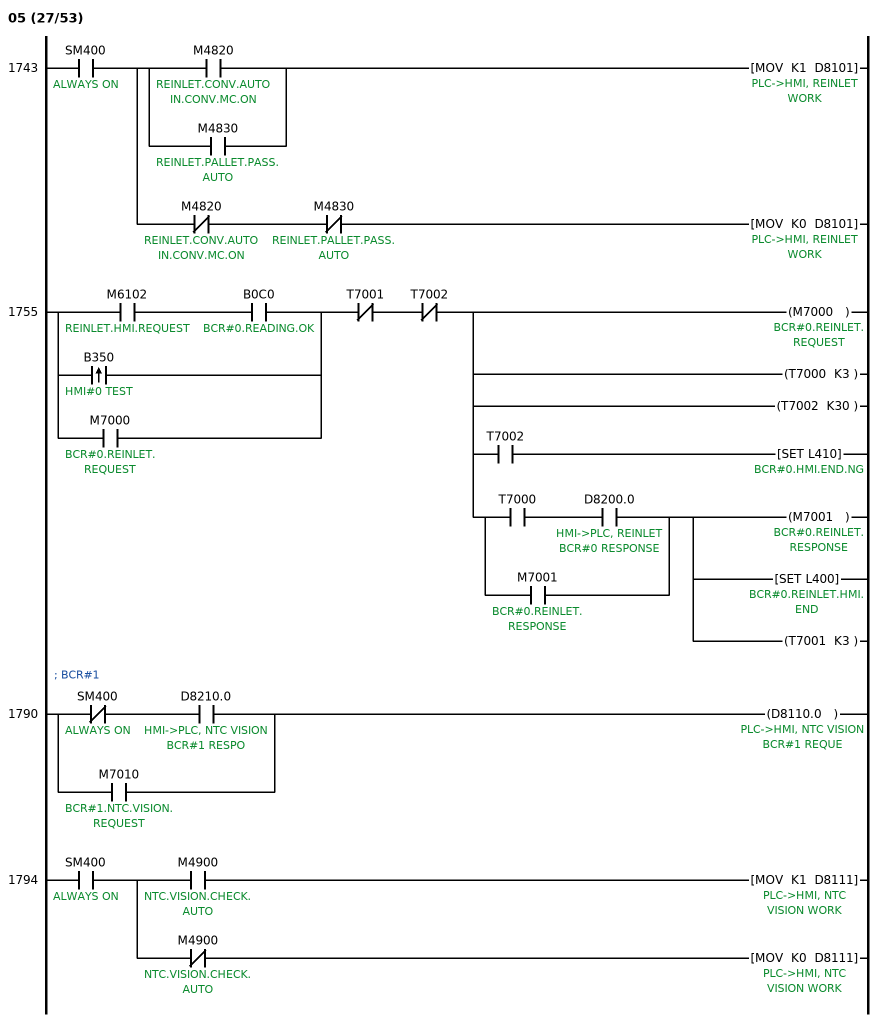
1743  LD      SM400  ; ALWAYS ON
      MPS
      LD      M4820  ; REINLET.CONV.AUTO IN.CONV.MC.ON
      OR      M4830  ; REINLET.PALLET.PASS.AUTO
      ANB
      MOV     K1 D8101  ; PLC->HMI, REINLET WORK
      MPP
      ANI     M4820  ; REINLET.CONV.AUTO IN.CONV.MC.ON
      ANI     M4830  ; REINLET.PALLET.PASS.AUTO
      MOV     K0 D8101
1755  LD      M6102  ; REINLET.HMI.REQUEST
      AND     B0C0  ; BCR#0.READING.OK
      ORP     B350  ; HMI#0 TEST
      OR      M7000  ; BCR#0.REINLET.REQUEST
      ANI     T7001
      ANI     T7002
      OUT     M7000  ; BCR#0.REINLET.REQUEST
      OUT     T7000 K3
      OUT     T7002 K30
      MPS
      AND     T7002
      SET     L410  ; BCR#0.HMI.END.NG
      MPP
      LD      T7000
      AND     D8200.0  ; HMI->PLC, REINLET BCR#0 RESPONSE
      OR      M7001  ; BCR#0.REINLET.RESPONSE
      ANB
      OUT     M7001  ; BCR#0.REINLET.RESPONSE
      SET     L400  ; BCR#0.REINLET.HMI.END
      OUT     T7001 K3
; BCR#1
1790  LDI     SM400  ; ALWAYS ON
      AND     D8210.0  ; HMI->PLC, NTC VISION BCR#1 RESPO
      OR      M7010  ; BCR#1.NTC.VISION.REQUEST
      OUT     D8110.0  ; PLC->HMI, NTC VISION BCR#1 REQUE
1794  LD      SM400  ; ALWAYS ON
      MPS
      AND     M4900  ; NTC.VISION.CHECK.AUTO
      MOV     K1 D8111  ; PLC->HMI, NTC VISION WORK
      MPP
      ANI     M4900  ; NTC.VISION.CHECK.AUTO
      MOV     K0 D8111
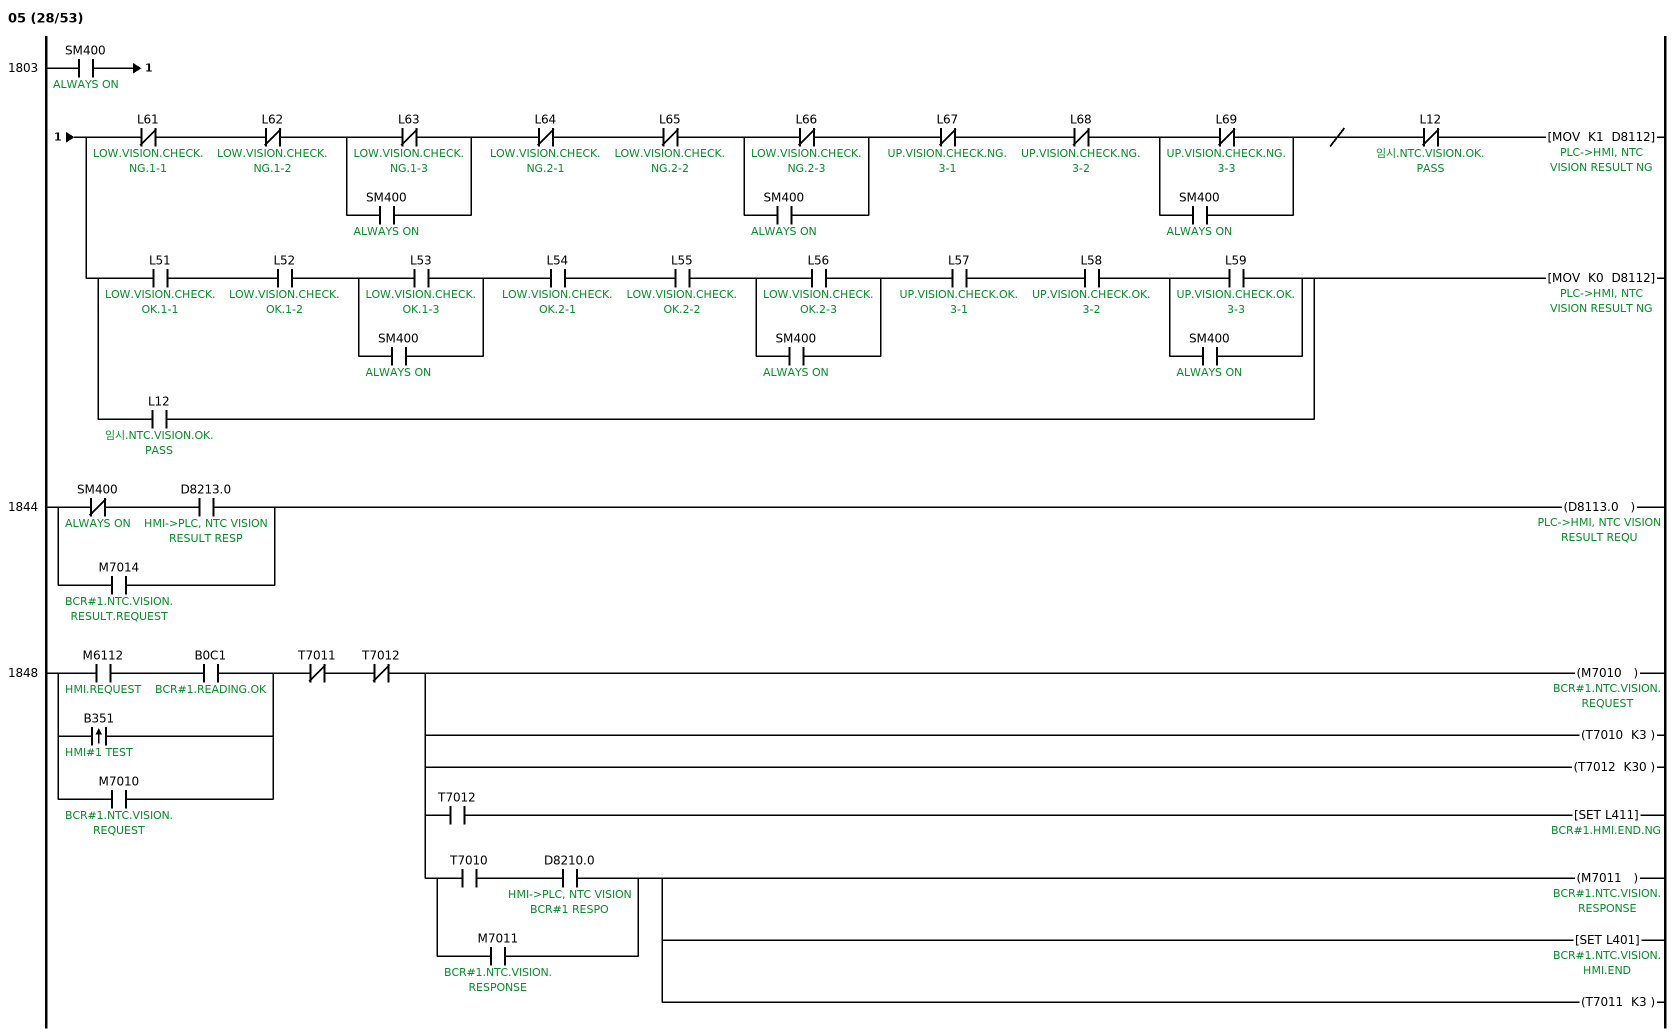
1803  LD      SM400  ; ALWAYS ON
      MPS
      ANI     L61  ; LOW.VISION.CHECK.NG.1-1
      ANI     L62  ; LOW.VISION.CHECK.NG.1-2
      LDI     L63  ; LOW.VISION.CHECK.NG.1-3
      OR      SM400  ; ALWAYS ON
      ANB
      ANI     L64  ; LOW.VISION.CHECK.NG.2-1
      ANI     L65  ; LOW.VISION.CHECK.NG.2-2
      LDI     L66  ; LOW.VISION.CHECK.NG.2-3
      OR      SM400  ; ALWAYS ON
      ANB
      ANI     L67  ; UP.VISION.CHECK.NG.3-1
      ANI     L68  ; UP.VISION.CHECK.NG.3-2
      LDI     L69  ; UP.VISION.CHECK.NG.3-3
      OR      SM400  ; ALWAYS ON
      ANB
      INV
      ANI     L12  ; 임시.NTC.VISION.OK.PASS
      MOV     K1 D8112  ; PLC->HMI, NTC VISION RESULT NG
      MPP
      LD      L51  ; LOW.VISION.CHECK.OK.1-1
      AND     L52  ; LOW.VISION.CHECK.OK.1-2
      LD      L53  ; LOW.VISION.CHECK.OK.1-3
      OR      SM400  ; ALWAYS ON
      ANB
      AND     L54  ; LOW.VISION.CHECK.OK.2-1
      AND     L55  ; LOW.VISION.CHECK.OK.2-2
      LD      L56  ; LOW.VISION.CHECK.OK.2-3
      OR      SM400  ; ALWAYS ON
      ANB
      AND     L57  ; UP.VISION.CHECK.OK.3-1
      AND     L58  ; UP.VISION.CHECK.OK.3-2
      LD      L59  ; UP.VISION.CHECK.OK.3-3
      OR      SM400  ; ALWAYS ON
      ANB
      OR      L12  ; 임시.NTC.VISION.OK.PASS
      ANB
      MOV     K0 D8112
1844  LDI     SM400  ; ALWAYS ON
      AND     D8213.0  ; HMI->PLC, NTC VISION RESULT RESP
      OR      M7014  ; BCR#1.NTC.VISION.RESULT.REQUEST
      OUT     D8113.0  ; PLC->HMI, NTC VISION RESULT REQU
1848  LD      M6112  ; HMI.REQUEST
      AND     B0C1  ; BCR#1.READING.OK
      ORP     B351  ; HMI#1 TEST
      OR      M7010  ; BCR#1.NTC.VISION.REQUEST
      ANI     T7011
      ANI     T7012
      OUT     M7010  ; BCR#1.NTC.VISION.REQUEST
      OUT     T7010 K3
      OUT     T7012 K30
      MPS
      AND     T7012
      SET     L411  ; BCR#1.HMI.END.NG
      MPP
      LD      T7010
      AND     D8210.0  ; HMI->PLC, NTC VISION BCR#1 RESPO
      OR      M7011  ; BCR#1.NTC.VISION.RESPONSE
      ANB
      OUT     M7011  ; BCR#1.NTC.VISION.RESPONSE
      SET     L401  ; BCR#1.NTC.VISION.HMI.END
      OUT     T7011 K3
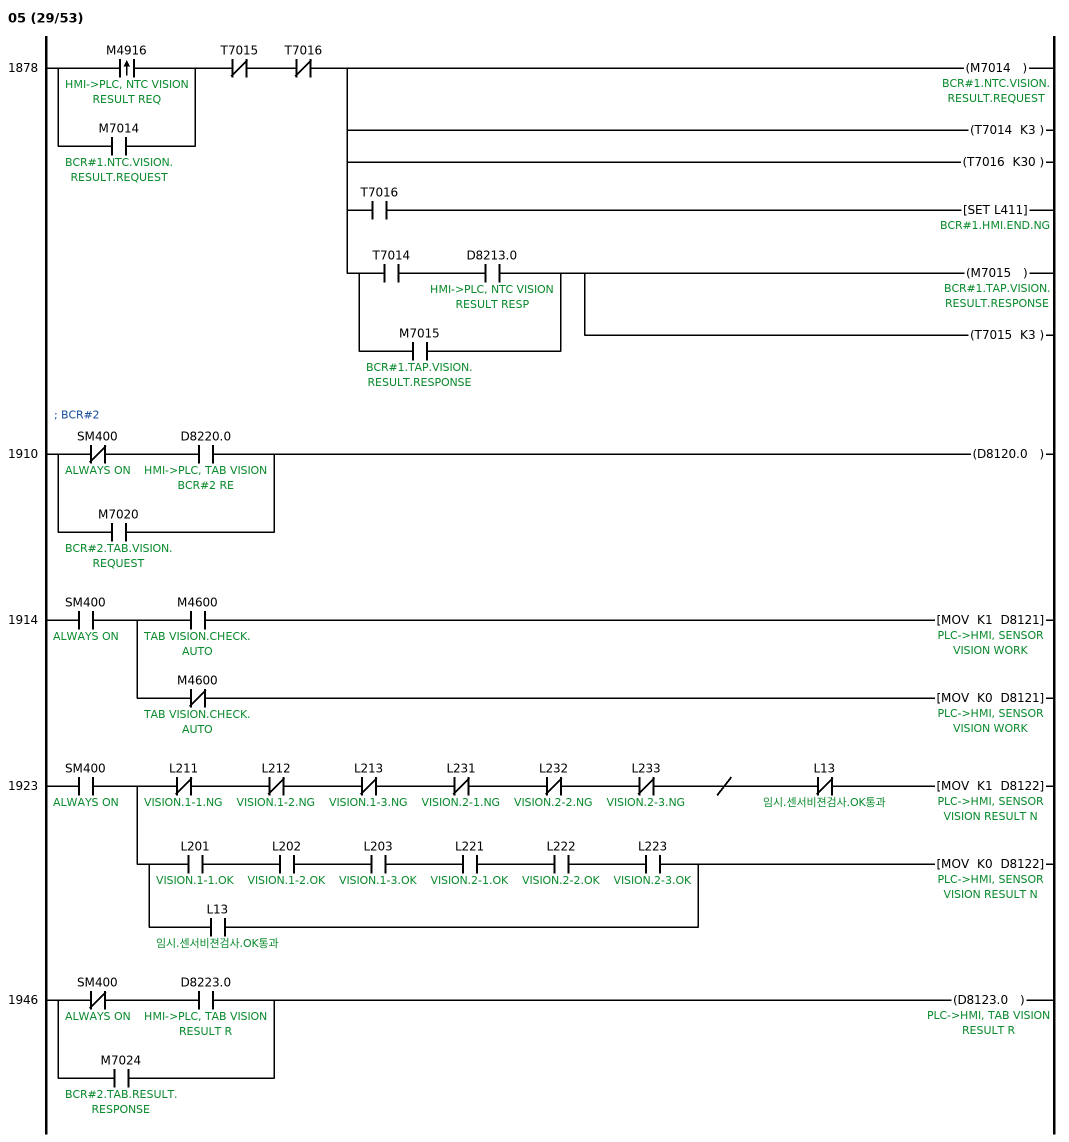
1878  LDP     M4916  ; HMI->PLC, NTC VISION RESULT REQ
      OR      M7014  ; BCR#1.NTC.VISION.RESULT.REQUEST
      ANI     T7015
      ANI     T7016
      OUT     M7014  ; BCR#1.NTC.VISION.RESULT.REQUEST
      OUT     T7014 K3
      OUT     T7016 K30
      MPS
      AND     T7016
      SET     L411  ; BCR#1.HMI.END.NG
      MPP
      LD      T7014
      AND     D8213.0  ; HMI->PLC, NTC VISION RESULT RESP
      OR      M7015  ; BCR#1.TAP.VISION.RESULT.RESPONSE
      ANB
      OUT     M7015  ; BCR#1.TAP.VISION.RESULT.RESPONSE
      OUT     T7015 K3
; BCR#2
1910  LDI     SM400  ; ALWAYS ON
      AND     D8220.0  ; HMI->PLC, TAB VISION BCR#2 RE
      OR      M7020  ; BCR#2.TAB.VISION.REQUEST
      OUT     D8120.0
1914  LD      SM400  ; ALWAYS ON
      MPS
      AND     M4600  ; TAB VISION.CHECK.AUTO
      MOV     K1 D8121  ; PLC->HMI, SENSOR VISION WORK
      MPP
      ANI     M4600  ; TAB VISION.CHECK.AUTO
      MOV     K0 D8121
1923  LD      SM400  ; ALWAYS ON
      MPS
      ANI     L211  ; VISION.1-1.NG
      ANI     L212  ; VISION.1-2.NG
      ANI     L213  ; VISION.1-3.NG
      ANI     L231  ; VISION.2-1.NG
      ANI     L232  ; VISION.2-2.NG
      ANI     L233  ; VISION.2-3.NG
      INV
      ANI     L13  ; 임시.센서비젼검사.OK통과
      MOV     K1 D8122  ; PLC->HMI, SENSOR VISION RESULT N
      MPP
      LD      L201  ; VISION.1-1.OK
      AND     L202  ; VISION.1-2.OK
      AND     L203  ; VISION.1-3.OK
      AND     L221  ; VISION.2-1.OK
      AND     L222  ; VISION.2-2.OK
      AND     L223  ; VISION.2-3.OK
      OR      L13  ; 임시.센서비젼검사.OK통과
      ANB
      MOV     K0 D8122
1946  LDI     SM400  ; ALWAYS ON
      AND     D8223.0  ; HMI->PLC, TAB VISION RESULT R
      OR      M7024  ; BCR#2.TAB.RESULT.RESPONSE
      OUT     D8123.0  ; PLC->HMI, TAB VISION RESULT R
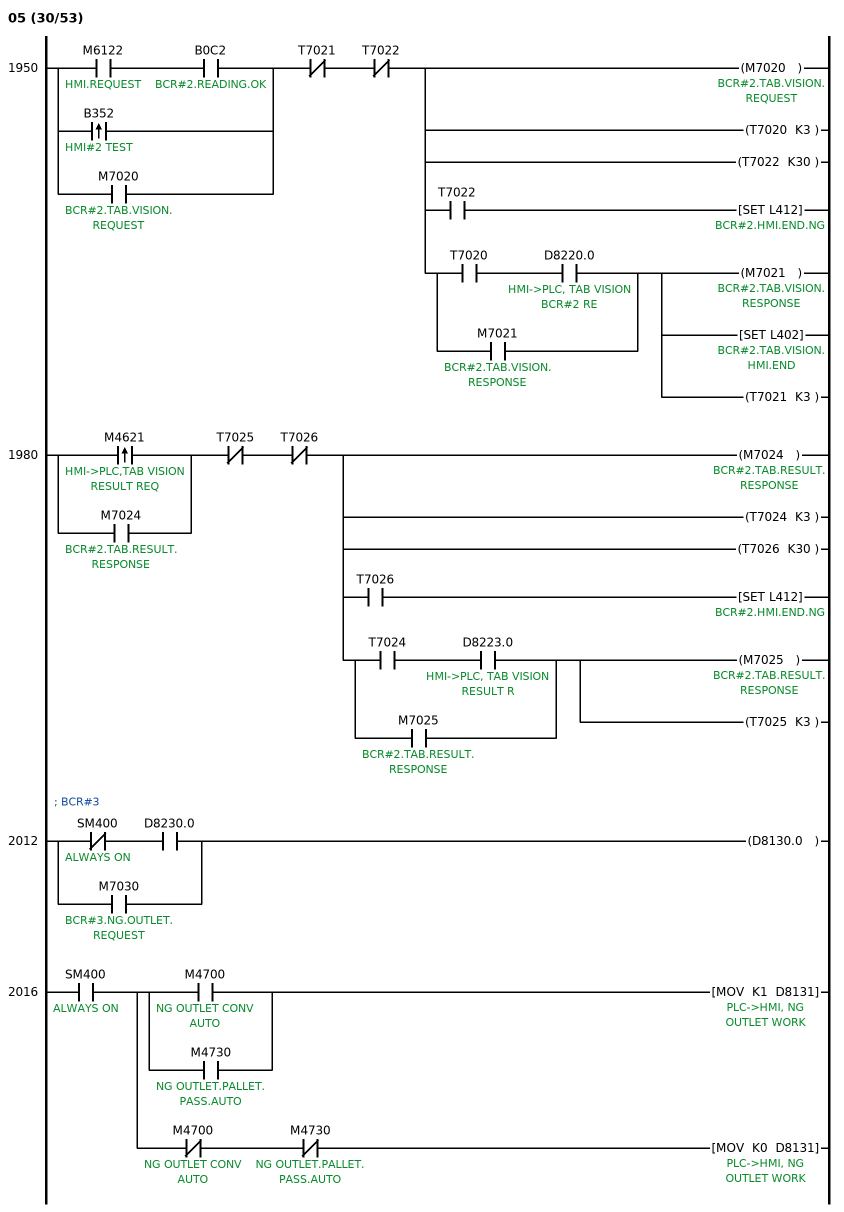
1950  LD      M6122  ; HMI.REQUEST
      AND     B0C2  ; BCR#2.READING.OK
      ORP     B352  ; HMI#2 TEST
      OR      M7020  ; BCR#2.TAB.VISION.REQUEST
      ANI     T7021
      ANI     T7022
      OUT     M7020  ; BCR#2.TAB.VISION.REQUEST
      OUT     T7020 K3
      OUT     T7022 K30
      MPS
      AND     T7022
      SET     L412  ; BCR#2.HMI.END.NG
      MPP
      LD      T7020
      AND     D8220.0  ; HMI->PLC, TAB VISION BCR#2 RE
      OR      M7021  ; BCR#2.TAB.VISION.RESPONSE
      ANB
      OUT     M7021  ; BCR#2.TAB.VISION.RESPONSE
      SET     L402  ; BCR#2.TAB.VISION.HMI.END
      OUT     T7021 K3
1980  LDP     M4621  ; HMI->PLC,TAB VISION RESULT REQ
      OR      M7024  ; BCR#2.TAB.RESULT.RESPONSE
      ANI     T7025
      ANI     T7026
      OUT     M7024  ; BCR#2.TAB.RESULT.RESPONSE
      OUT     T7024 K3
      OUT     T7026 K30
      MPS
      AND     T7026
      SET     L412  ; BCR#2.HMI.END.NG
      MPP
      LD      T7024
      AND     D8223.0  ; HMI->PLC, TAB VISION RESULT R
      OR      M7025  ; BCR#2.TAB.RESULT.RESPONSE
      ANB
      OUT     M7025  ; BCR#2.TAB.RESULT.RESPONSE
      OUT     T7025 K3
; BCR#3
2012  LDI     SM400  ; ALWAYS ON
      AND     D8230.0
      OR      M7030  ; BCR#3.NG.OUTLET.REQUEST
      OUT     D8130.0
2016  LD      SM400  ; ALWAYS ON
      MPS
      LD      M4700  ; NG OUTLET CONV AUTO
      OR      M4730  ; NG OUTLET.PALLET.PASS.AUTO
      ANB
      MOV     K1 D8131  ; PLC->HMI, NG OUTLET WORK
      MPP
      ANI     M4700  ; NG OUTLET CONV AUTO
      ANI     M4730  ; NG OUTLET.PALLET.PASS.AUTO
      MOV     K0 D8131
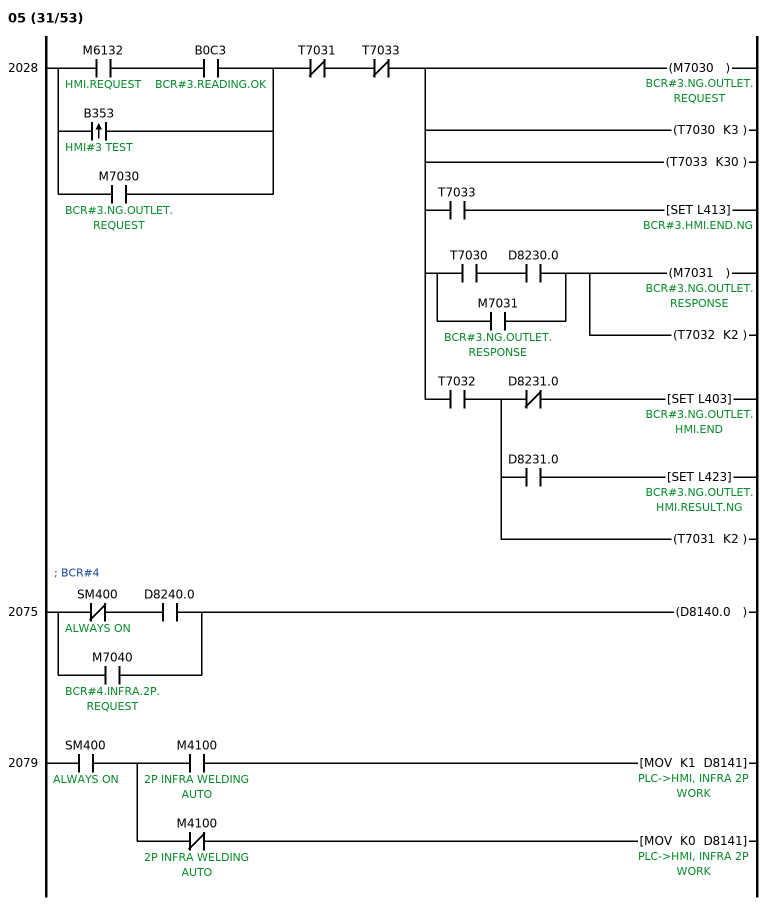
2028  LD      M6132  ; HMI.REQUEST
      AND     B0C3  ; BCR#3.READING.OK
      ORP     B353  ; HMI#3 TEST
      OR      M7030  ; BCR#3.NG.OUTLET.REQUEST
      ANI     T7031
      ANI     T7033
      OUT     M7030  ; BCR#3.NG.OUTLET.REQUEST
      OUT     T7030 K3
      OUT     T7033 K30
      MPS
      AND     T7033
      SET     L413  ; BCR#3.HMI.END.NG
      MRD
      LD      T7030
      AND     D8230.0
      OR      M7031  ; BCR#3.NG.OUTLET.RESPONSE
      ANB
      OUT     M7031  ; BCR#3.NG.OUTLET.RESPONSE
      OUT     T7032 K2
      MPP
      AND     T7032
      MPS
      ANI     D8231.0
      SET     L403  ; BCR#3.NG.OUTLET.HMI.END
      MRD
      AND     D8231.0
      SET     L423  ; BCR#3.NG.OUTLET.HMI.RESULT.NG
      MPP
      OUT     T7031 K2
; BCR#4
2075  LDI     SM400  ; ALWAYS ON
      AND     D8240.0
      OR      M7040  ; BCR#4.INFRA.2P.REQUEST
      OUT     D8140.0
2079  LD      SM400  ; ALWAYS ON
      MPS
      AND     M4100  ; 2P INFRA WELDING AUTO
      MOV     K1 D8141  ; PLC->HMI, INFRA 2P WORK
      MPP
      ANI     M4100  ; 2P INFRA WELDING AUTO
      MOV     K0 D8141
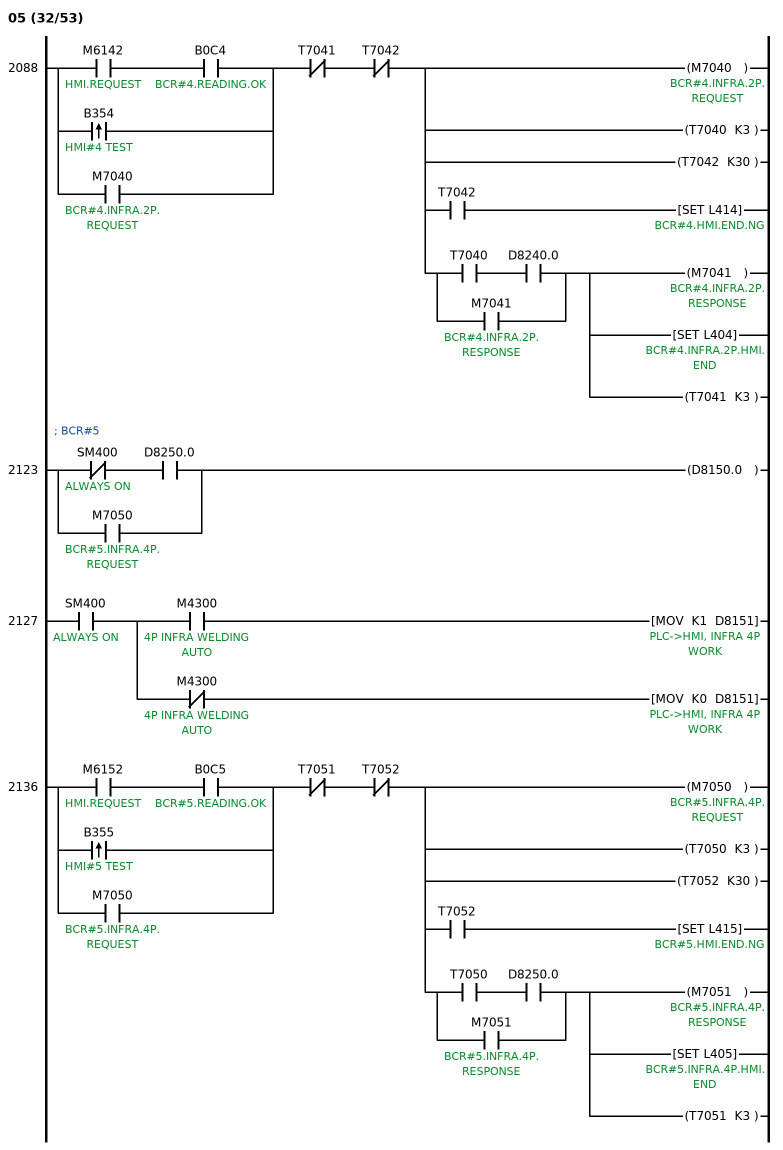
2088  LD      M6142  ; HMI.REQUEST
      AND     B0C4  ; BCR#4.READING.OK
      ORP     B354  ; HMI#4 TEST
      OR      M7040  ; BCR#4.INFRA.2P.REQUEST
      ANI     T7041
      ANI     T7042
      OUT     M7040  ; BCR#4.INFRA.2P.REQUEST
      OUT     T7040 K3
      OUT     T7042 K30
      MPS
      AND     T7042
      SET     L414  ; BCR#4.HMI.END.NG
      MPP
      LD      T7040
      AND     D8240.0
      OR      M7041  ; BCR#4.INFRA.2P.RESPONSE
      ANB
      OUT     M7041  ; BCR#4.INFRA.2P.RESPONSE
      SET     L404  ; BCR#4.INFRA.2P.HMI.END
      OUT     T7041 K3
; BCR#5
2123  LDI     SM400  ; ALWAYS ON
      AND     D8250.0
      OR      M7050  ; BCR#5.INFRA.4P.REQUEST
      OUT     D8150.0
2127  LD      SM400  ; ALWAYS ON
      MPS
      AND     M4300  ; 4P INFRA WELDING AUTO
      MOV     K1 D8151  ; PLC->HMI, INFRA 4P WORK
      MPP
      ANI     M4300  ; 4P INFRA WELDING AUTO
      MOV     K0 D8151
2136  LD      M6152  ; HMI.REQUEST
      AND     B0C5  ; BCR#5.READING.OK
      ORP     B355  ; HMI#5 TEST
      OR      M7050  ; BCR#5.INFRA.4P.REQUEST
      ANI     T7051
      ANI     T7052
      OUT     M7050  ; BCR#5.INFRA.4P.REQUEST
      OUT     T7050 K3
      OUT     T7052 K30
      MPS
      AND     T7052
      SET     L415  ; BCR#5.HMI.END.NG
      MPP
      LD      T7050
      AND     D8250.0
      OR      M7051  ; BCR#5.INFRA.4P.RESPONSE
      ANB
      OUT     M7051  ; BCR#5.INFRA.4P.RESPONSE
      SET     L405  ; BCR#5.INFRA.4P.HMI.END
      OUT     T7051 K3
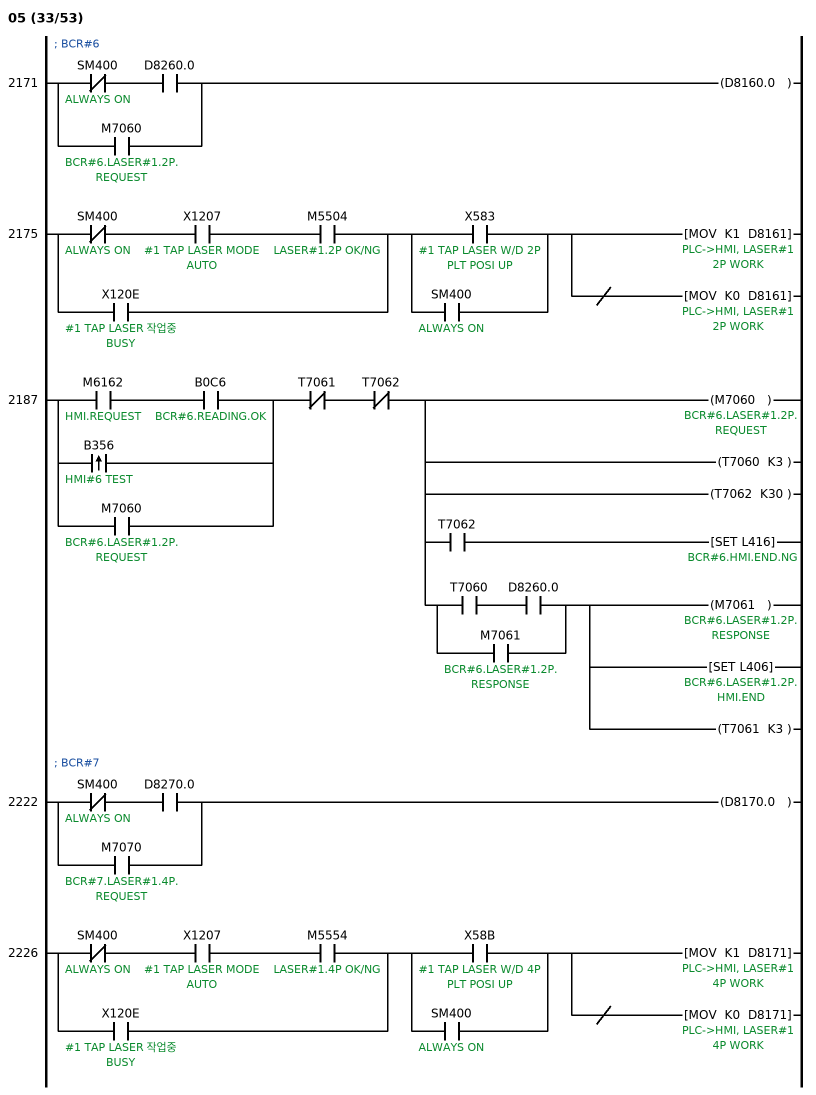
; BCR#6
2171  LDI     SM400  ; ALWAYS ON
      AND     D8260.0
      OR      M7060  ; BCR#6.LASER#1.2P.REQUEST
      OUT     D8160.0
2175  LDI     SM400  ; ALWAYS ON
      AND     X1207  ; #1 TAP LASER MODE AUTO
      AND     M5504  ; LASER#1.2P OK/NG
      OR      X120E  ; #1 TAP LASER 작업중 BUSY
      LD      X583  ; #1 TAP LASER W/D 2P PLT POSI UP
      OR      SM400  ; ALWAYS ON
      ANB
      MOV     K1 D8161  ; PLC->HMI, LASER#1 2P WORK
      INV
      MOV     K0 D8161
2187  LD      M6162  ; HMI.REQUEST
      AND     B0C6  ; BCR#6.READING.OK
      ORP     B356  ; HMI#6 TEST
      OR      M7060  ; BCR#6.LASER#1.2P.REQUEST
      ANI     T7061
      ANI     T7062
      OUT     M7060  ; BCR#6.LASER#1.2P.REQUEST
      OUT     T7060 K3
      OUT     T7062 K30
      MPS
      AND     T7062
      SET     L416  ; BCR#6.HMI.END.NG
      MPP
      LD      T7060
      AND     D8260.0
      OR      M7061  ; BCR#6.LASER#1.2P.RESPONSE
      ANB
      OUT     M7061  ; BCR#6.LASER#1.2P.RESPONSE
      SET     L406  ; BCR#6.LASER#1.2P.HMI.END
      OUT     T7061 K3
; BCR#7
2222  LDI     SM400  ; ALWAYS ON
      AND     D8270.0
      OR      M7070  ; BCR#7.LASER#1.4P.REQUEST
      OUT     D8170.0
2226  LDI     SM400  ; ALWAYS ON
      AND     X1207  ; #1 TAP LASER MODE AUTO
      AND     M5554  ; LASER#1.4P OK/NG
      OR      X120E  ; #1 TAP LASER 작업중 BUSY
      LD      X58B  ; #1 TAP LASER W/D 4P PLT POSI UP
      OR      SM400  ; ALWAYS ON
      ANB
      MOV     K1 D8171  ; PLC->HMI, LASER#1 4P WORK
      INV
      MOV     K0 D8171
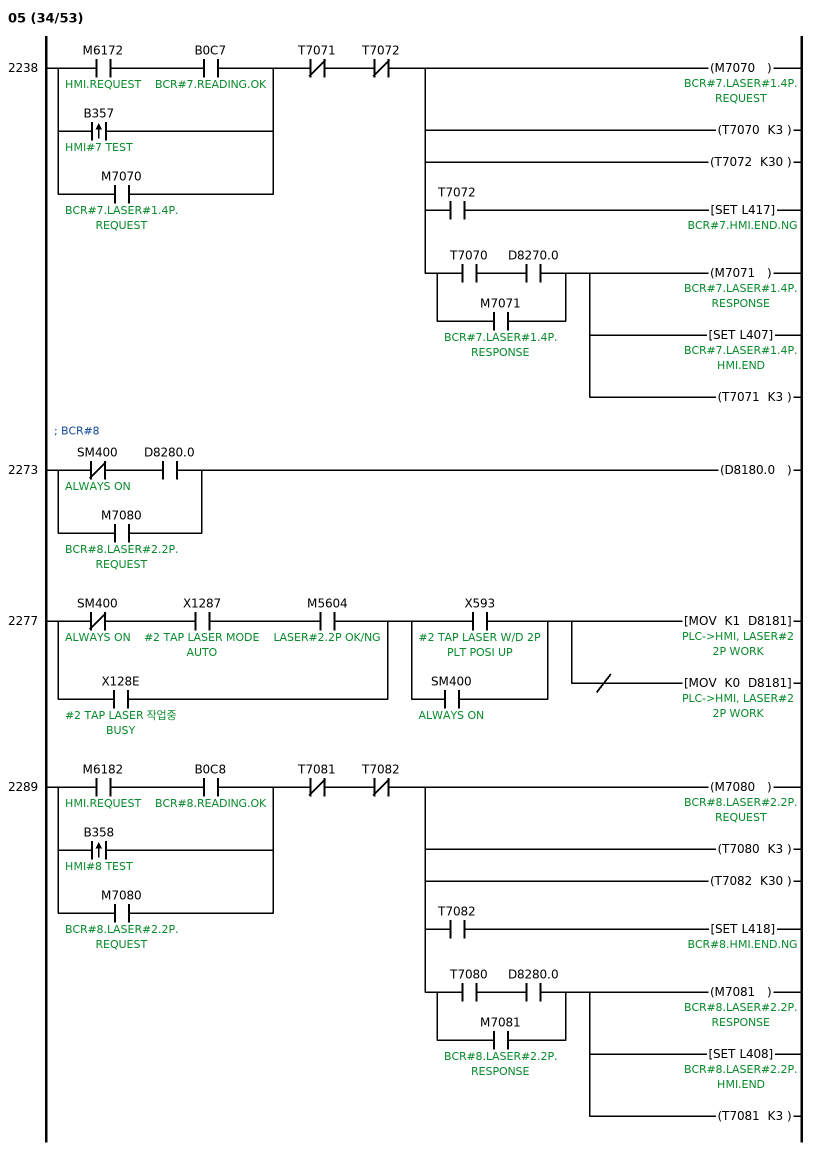
2238  LD      M6172  ; HMI.REQUEST
      AND     B0C7  ; BCR#7.READING.OK
      ORP     B357  ; HMI#7 TEST
      OR      M7070  ; BCR#7.LASER#1.4P.REQUEST
      ANI     T7071
      ANI     T7072
      OUT     M7070  ; BCR#7.LASER#1.4P.REQUEST
      OUT     T7070 K3
      OUT     T7072 K30
      MPS
      AND     T7072
      SET     L417  ; BCR#7.HMI.END.NG
      MPP
      LD      T7070
      AND     D8270.0
      OR      M7071  ; BCR#7.LASER#1.4P.RESPONSE
      ANB
      OUT     M7071  ; BCR#7.LASER#1.4P.RESPONSE
      SET     L407  ; BCR#7.LASER#1.4P.HMI.END
      OUT     T7071 K3
; BCR#8
2273  LDI     SM400  ; ALWAYS ON
      AND     D8280.0
      OR      M7080  ; BCR#8.LASER#2.2P.REQUEST
      OUT     D8180.0
2277  LDI     SM400  ; ALWAYS ON
      AND     X1287  ; #2 TAP LASER MODE AUTO
      AND     M5604  ; LASER#2.2P OK/NG
      OR      X128E  ; #2 TAP LASER 작업중 BUSY
      LD      X593  ; #2 TAP LASER W/D 2P PLT POSI UP
      OR      SM400  ; ALWAYS ON
      ANB
      MOV     K1 D8181  ; PLC->HMI, LASER#2 2P WORK
      INV
      MOV     K0 D8181
2289  LD      M6182  ; HMI.REQUEST
      AND     B0C8  ; BCR#8.READING.OK
      ORP     B358  ; HMI#8 TEST
      OR      M7080  ; BCR#8.LASER#2.2P.REQUEST
      ANI     T7081
      ANI     T7082
      OUT     M7080  ; BCR#8.LASER#2.2P.REQUEST
      OUT     T7080 K3
      OUT     T7082 K30
      MPS
      AND     T7082
      SET     L418  ; BCR#8.HMI.END.NG
      MPP
      LD      T7080
      AND     D8280.0
      OR      M7081  ; BCR#8.LASER#2.2P.RESPONSE
      ANB
      OUT     M7081  ; BCR#8.LASER#2.2P.RESPONSE
      SET     L408  ; BCR#8.LASER#2.2P.HMI.END
      OUT     T7081 K3
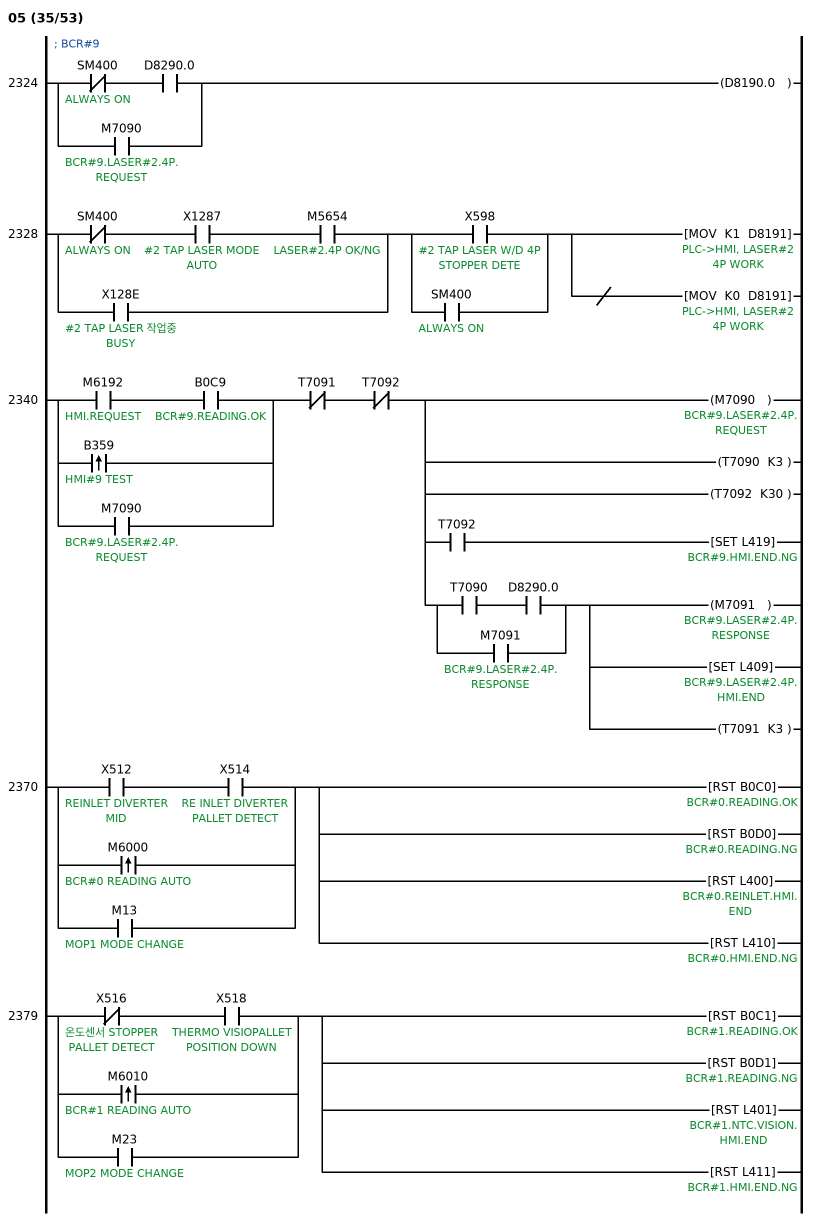
; BCR#9
2324  LDI     SM400  ; ALWAYS ON
      AND     D8290.0
      OR      M7090  ; BCR#9.LASER#2.4P.REQUEST
      OUT     D8190.0
2328  LDI     SM400  ; ALWAYS ON
      AND     X1287  ; #2 TAP LASER MODE AUTO
      AND     M5654  ; LASER#2.4P OK/NG
      OR      X128E  ; #2 TAP LASER 작업중 BUSY
      LD      X598  ; #2 TAP LASER W/D 4P STOPPER DETE
      OR      SM400  ; ALWAYS ON
      ANB
      MOV     K1 D8191  ; PLC->HMI, LASER#2 4P WORK
      INV
      MOV     K0 D8191
2340  LD      M6192  ; HMI.REQUEST
      AND     B0C9  ; BCR#9.READING.OK
      ORP     B359  ; HMI#9 TEST
      OR      M7090  ; BCR#9.LASER#2.4P.REQUEST
      ANI     T7091
      ANI     T7092
      OUT     M7090  ; BCR#9.LASER#2.4P.REQUEST
      OUT     T7090 K3
      OUT     T7092 K30
      MPS
      AND     T7092
      SET     L419  ; BCR#9.HMI.END.NG
      MPP
      LD      T7090
      AND     D8290.0
      OR      M7091  ; BCR#9.LASER#2.4P.RESPONSE
      ANB
      OUT     M7091  ; BCR#9.LASER#2.4P.RESPONSE
      SET     L409  ; BCR#9.LASER#2.4P.HMI.END
      OUT     T7091 K3
2370  LD      X512  ; REINLET DIVERTER MID
      AND     X514  ; RE INLET DIVERTER PALLET DETECT
      ORP     M6000  ; BCR#0 READING AUTO
      OR      M13  ; MOP1 MODE CHANGE
      RST     B0C0  ; BCR#0.READING.OK
      RST     B0D0  ; BCR#0.READING.NG
      RST     L400  ; BCR#0.REINLET.HMI.END
      RST     L410  ; BCR#0.HMI.END.NG
2379  LDI     X516  ; 온도센서 STOPPER PALLET DETECT
      AND     X518  ; THERMO VISIOPALLET POSITION DOWN
      ORP     M6010  ; BCR#1 READING AUTO
      OR      M23  ; MOP2 MODE CHANGE
      RST     B0C1  ; BCR#1.READING.OK
      RST     B0D1  ; BCR#1.READING.NG
      RST     L401  ; BCR#1.NTC.VISION.HMI.END
      RST     L411  ; BCR#1.HMI.END.NG
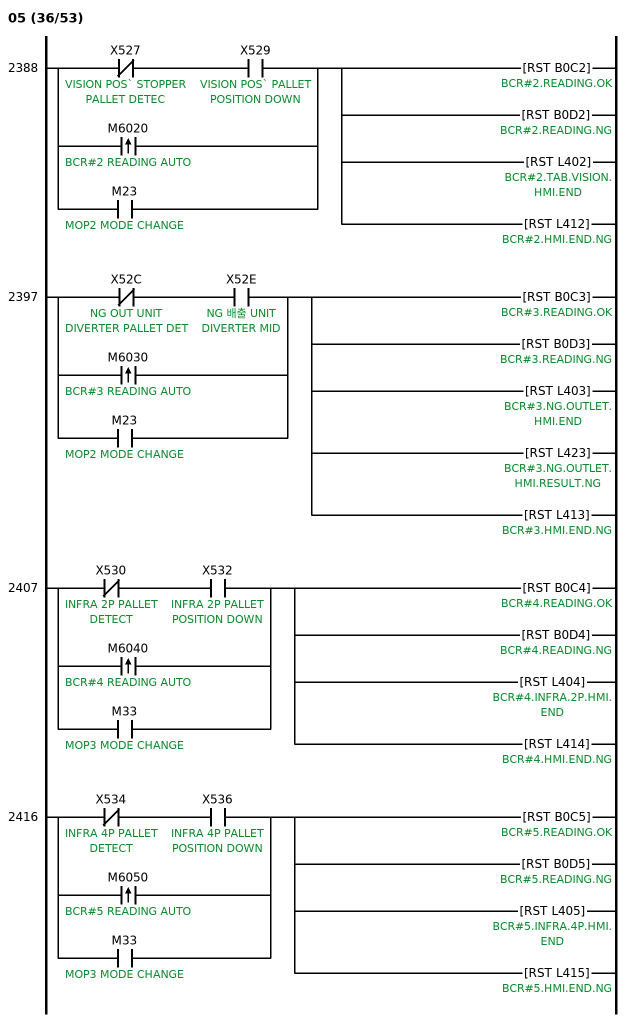
2388  LDI     X527  ; VISION POS` STOPPER PALLET DETEC
      AND     X529  ; VISION POS` PALLET POSITION DOWN
      ORP     M6020  ; BCR#2 READING AUTO
      OR      M23  ; MOP2 MODE CHANGE
      RST     B0C2  ; BCR#2.READING.OK
      RST     B0D2  ; BCR#2.READING.NG
      RST     L402  ; BCR#2.TAB.VISION.HMI.END
      RST     L412  ; BCR#2.HMI.END.NG
2397  LDI     X52C  ; NG OUT UNIT DIVERTER PALLET DET
      AND     X52E  ; NG 배출 UNIT DIVERTER MID
      ORP     M6030  ; BCR#3 READING AUTO
      OR      M23  ; MOP2 MODE CHANGE
      RST     B0C3  ; BCR#3.READING.OK
      RST     B0D3  ; BCR#3.READING.NG
      RST     L403  ; BCR#3.NG.OUTLET.HMI.END
      RST     L423  ; BCR#3.NG.OUTLET.HMI.RESULT.NG
      RST     L413  ; BCR#3.HMI.END.NG
2407  LDI     X530  ; INFRA 2P PALLET DETECT
      AND     X532  ; INFRA 2P PALLET POSITION DOWN
      ORP     M6040  ; BCR#4 READING AUTO
      OR      M33  ; MOP3 MODE CHANGE
      RST     B0C4  ; BCR#4.READING.OK
      RST     B0D4  ; BCR#4.READING.NG
      RST     L404  ; BCR#4.INFRA.2P.HMI.END
      RST     L414  ; BCR#4.HMI.END.NG
2416  LDI     X534  ; INFRA 4P PALLET DETECT
      AND     X536  ; INFRA 4P PALLET POSITION DOWN
      ORP     M6050  ; BCR#5 READING AUTO
      OR      M33  ; MOP3 MODE CHANGE
      RST     B0C5  ; BCR#5.READING.OK
      RST     B0D5  ; BCR#5.READING.NG
      RST     L405  ; BCR#5.INFRA.4P.HMI.END
      RST     L415  ; BCR#5.HMI.END.NG
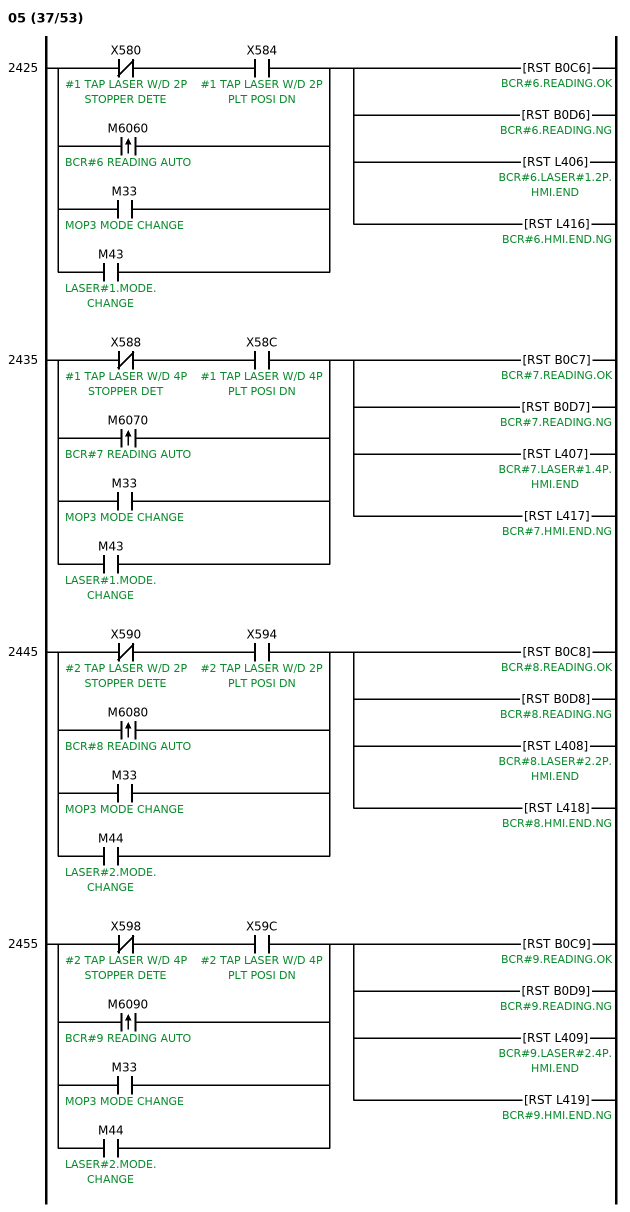
2425  LDI     X580  ; #1 TAP LASER W/D 2P STOPPER DETE
      AND     X584  ; #1 TAP LASER W/D 2P PLT POSI DN
      ORP     M6060  ; BCR#6 READING AUTO
      OR      M33  ; MOP3 MODE CHANGE
      OR      M43  ; LASER#1.MODE.CHANGE
      RST     B0C6  ; BCR#6.READING.OK
      RST     B0D6  ; BCR#6.READING.NG
      RST     L406  ; BCR#6.LASER#1.2P.HMI.END
      RST     L416  ; BCR#6.HMI.END.NG
2435  LDI     X588  ; #1 TAP LASER W/D 4P STOPPER DET
      AND     X58C  ; #1 TAP LASER W/D 4P PLT POSI DN
      ORP     M6070  ; BCR#7 READING AUTO
      OR      M33  ; MOP3 MODE CHANGE
      OR      M43  ; LASER#1.MODE.CHANGE
      RST     B0C7  ; BCR#7.READING.OK
      RST     B0D7  ; BCR#7.READING.NG
      RST     L407  ; BCR#7.LASER#1.4P.HMI.END
      RST     L417  ; BCR#7.HMI.END.NG
2445  LDI     X590  ; #2 TAP LASER W/D 2P STOPPER DETE
      AND     X594  ; #2 TAP LASER W/D 2P PLT POSI DN
      ORP     M6080  ; BCR#8 READING AUTO
      OR      M33  ; MOP3 MODE CHANGE
      OR      M44  ; LASER#2.MODE.CHANGE
      RST     B0C8  ; BCR#8.READING.OK
      RST     B0D8  ; BCR#8.READING.NG
      RST     L408  ; BCR#8.LASER#2.2P.HMI.END
      RST     L418  ; BCR#8.HMI.END.NG
2455  LDI     X598  ; #2 TAP LASER W/D 4P STOPPER DETE
      AND     X59C  ; #2 TAP LASER W/D 4P PLT POSI DN
      ORP     M6090  ; BCR#9 READING AUTO
      OR      M33  ; MOP3 MODE CHANGE
      OR      M44  ; LASER#2.MODE.CHANGE
      RST     B0C9  ; BCR#9.READING.OK
      RST     B0D9  ; BCR#9.READING.NG
      RST     L409  ; BCR#9.LASER#2.4P.HMI.END
      RST     L419  ; BCR#9.HMI.END.NG
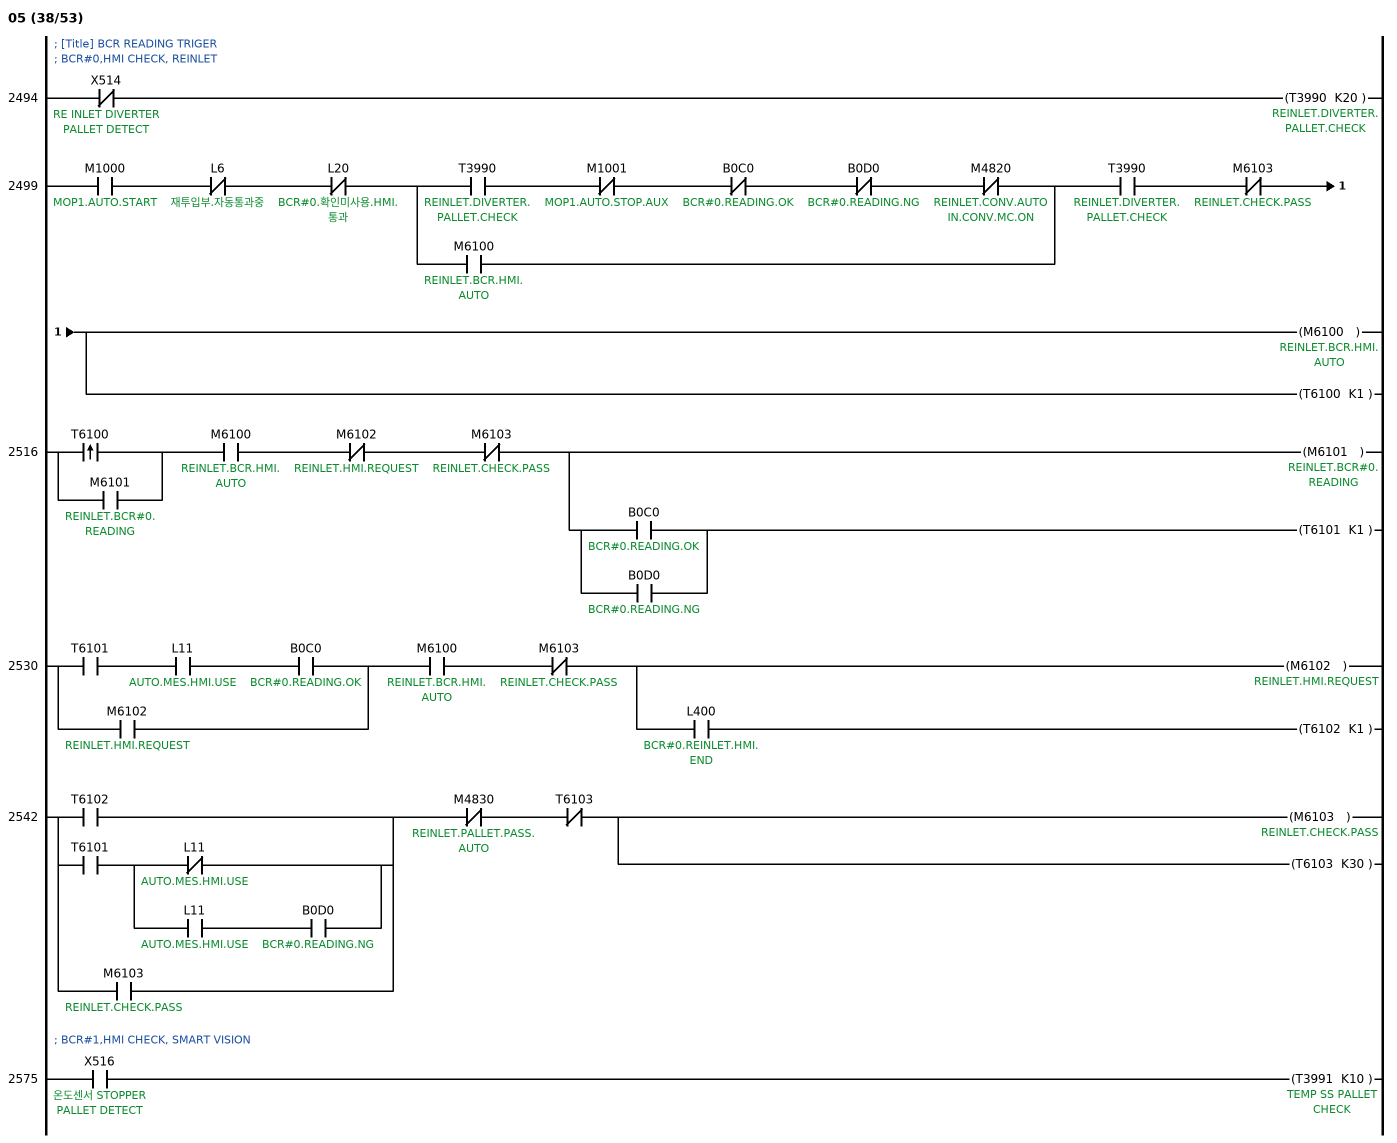
; [Title] BCR READING TRIGER
; BCR#0,HMI CHECK, REINLET
2494  LDI     X514  ; RE INLET DIVERTER PALLET DETECT
      OUT     T3990 K20  ; REINLET.DIVERTER.PALLET.CHECK
2499  LD      M1000  ; MOP1.AUTO.START
      ANI     L6  ; 재투입부.자동통과중
      ANI     L20  ; BCR#0.확인미사용.HMI.통과
      LD      T3990  ; REINLET.DIVERTER.PALLET.CHECK
      ANI     M1001  ; MOP1.AUTO.STOP.AUX
      ANI     B0C0  ; BCR#0.READING.OK
      ANI     B0D0  ; BCR#0.READING.NG
      ANI     M4820  ; REINLET.CONV.AUTO IN.CONV.MC.ON
      OR      M6100  ; REINLET.BCR.HMI.AUTO
      ANB
      AND     T3990  ; REINLET.DIVERTER.PALLET.CHECK
      ANI     M6103  ; REINLET.CHECK.PASS
      OUT     M6100  ; REINLET.BCR.HMI.AUTO
      OUT     T6100 K1
2516  LDP     T6100
      OR      M6101  ; REINLET.BCR#0.READING
      AND     M6100  ; REINLET.BCR.HMI.AUTO
      ANI     M6102  ; REINLET.HMI.REQUEST
      ANI     M6103  ; REINLET.CHECK.PASS
      OUT     M6101  ; REINLET.BCR#0.READING
      LD      B0C0  ; BCR#0.READING.OK
      OR      B0D0  ; BCR#0.READING.NG
      ANB
      OUT     T6101 K1
2530  LD      T6101
      AND     L11  ; AUTO.MES.HMI.USE
      AND     B0C0  ; BCR#0.READING.OK
      OR      M6102  ; REINLET.HMI.REQUEST
      AND     M6100  ; REINLET.BCR.HMI.AUTO
      ANI     M6103  ; REINLET.CHECK.PASS
      OUT     M6102  ; REINLET.HMI.REQUEST
      AND     L400  ; BCR#0.REINLET.HMI.END
      OUT     T6102 K1
2542  LD      T6102
      LD      T6101
      LDI     L11  ; AUTO.MES.HMI.USE
      LD      L11  ; AUTO.MES.HMI.USE
      AND     B0D0  ; BCR#0.READING.NG
      ORB
      ANB
      ORB
      OR      M6103  ; REINLET.CHECK.PASS
      ANI     M4830  ; REINLET.PALLET.PASS.AUTO
      ANI     T6103
      OUT     M6103  ; REINLET.CHECK.PASS
      OUT     T6103 K30
; BCR#1,HMI CHECK, SMART VISION
2575  LD      X516  ; 온도센서 STOPPER PALLET DETECT
      OUT     T3991 K10  ; TEMP SS PALLET CHECK
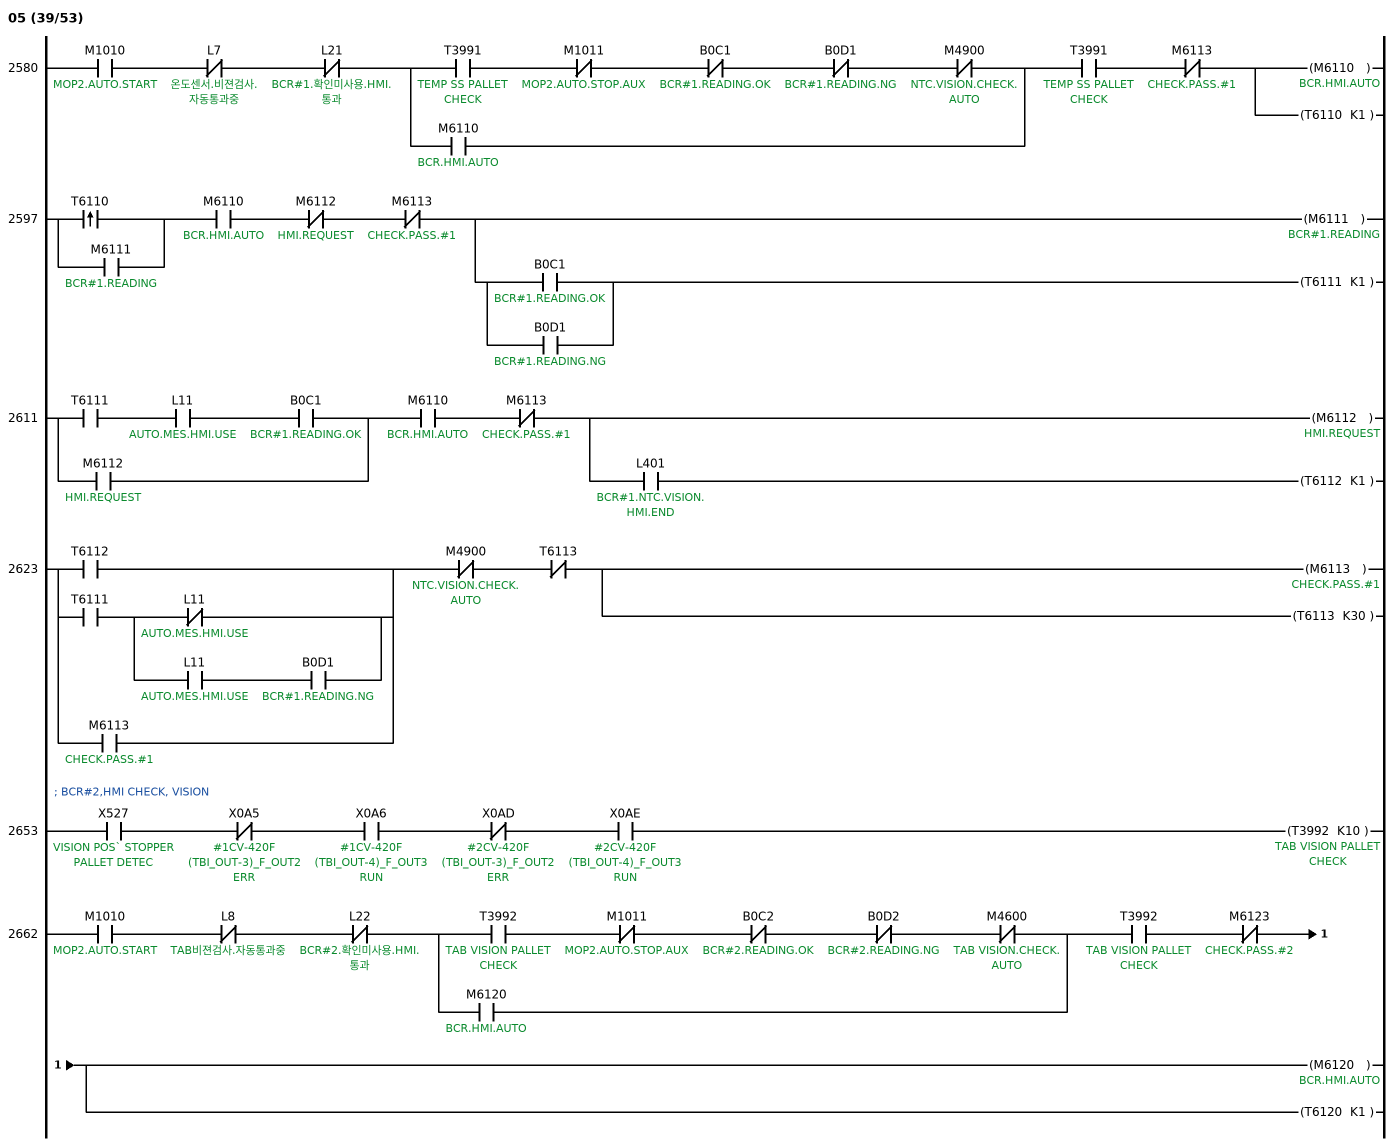
2580  LD      M1010  ; MOP2.AUTO.START
      ANI     L7  ; 온도센서.비젼검사.자동통과중
      ANI     L21  ; BCR#1.확인미사용.HMI.통과
      LD      T3991  ; TEMP SS PALLET CHECK
      ANI     M1011  ; MOP2.AUTO.STOP.AUX
      ANI     B0C1  ; BCR#1.READING.OK
      ANI     B0D1  ; BCR#1.READING.NG
      ANI     M4900  ; NTC.VISION.CHECK.AUTO
      OR      M6110  ; BCR.HMI.AUTO
      ANB
      AND     T3991  ; TEMP SS PALLET CHECK
      ANI     M6113  ; CHECK.PASS.#1
      OUT     M6110  ; BCR.HMI.AUTO
      OUT     T6110 K1
2597  LDP     T6110
      OR      M6111  ; BCR#1.READING
      AND     M6110  ; BCR.HMI.AUTO
      ANI     M6112  ; HMI.REQUEST
      ANI     M6113  ; CHECK.PASS.#1
      OUT     M6111  ; BCR#1.READING
      LD      B0C1  ; BCR#1.READING.OK
      OR      B0D1  ; BCR#1.READING.NG
      ANB
      OUT     T6111 K1
2611  LD      T6111
      AND     L11  ; AUTO.MES.HMI.USE
      AND     B0C1  ; BCR#1.READING.OK
      OR      M6112  ; HMI.REQUEST
      AND     M6110  ; BCR.HMI.AUTO
      ANI     M6113  ; CHECK.PASS.#1
      OUT     M6112  ; HMI.REQUEST
      AND     L401  ; BCR#1.NTC.VISION.HMI.END
      OUT     T6112 K1
2623  LD      T6112
      LD      T6111
      LDI     L11  ; AUTO.MES.HMI.USE
      LD      L11  ; AUTO.MES.HMI.USE
      AND     B0D1  ; BCR#1.READING.NG
      ORB
      ANB
      ORB
      OR      M6113  ; CHECK.PASS.#1
      ANI     M4900  ; NTC.VISION.CHECK.AUTO
      ANI     T6113
      OUT     M6113  ; CHECK.PASS.#1
      OUT     T6113 K30
; BCR#2,HMI CHECK, VISION
2653  LD      X527  ; VISION POS` STOPPER PALLET DETEC
      ANI     X0A5  ; #1CV-420F (TBI_OUT-3)_F_OUT2 ERR
      AND     X0A6  ; #1CV-420F (TBI_OUT-4)_F_OUT3 RUN
      ANI     X0AD  ; #2CV-420F (TBI_OUT-3)_F_OUT2 ERR
      AND     X0AE  ; #2CV-420F (TBI_OUT-4)_F_OUT3 RUN
      OUT     T3992 K10  ; TAB VISION PALLET CHECK
2662  LD      M1010  ; MOP2.AUTO.START
      ANI     L8  ; TAB비젼검사.자동통과중
      ANI     L22  ; BCR#2.확인미사용.HMI.통과
      LD      T3992  ; TAB VISION PALLET CHECK
      ANI     M1011  ; MOP2.AUTO.STOP.AUX
      ANI     B0C2  ; BCR#2.READING.OK
      ANI     B0D2  ; BCR#2.READING.NG
      ANI     M4600  ; TAB VISION.CHECK.AUTO
      OR      M6120  ; BCR.HMI.AUTO
      ANB
      AND     T3992  ; TAB VISION PALLET CHECK
      ANI     M6123  ; CHECK.PASS.#2
      OUT     M6120  ; BCR.HMI.AUTO
      OUT     T6120 K1
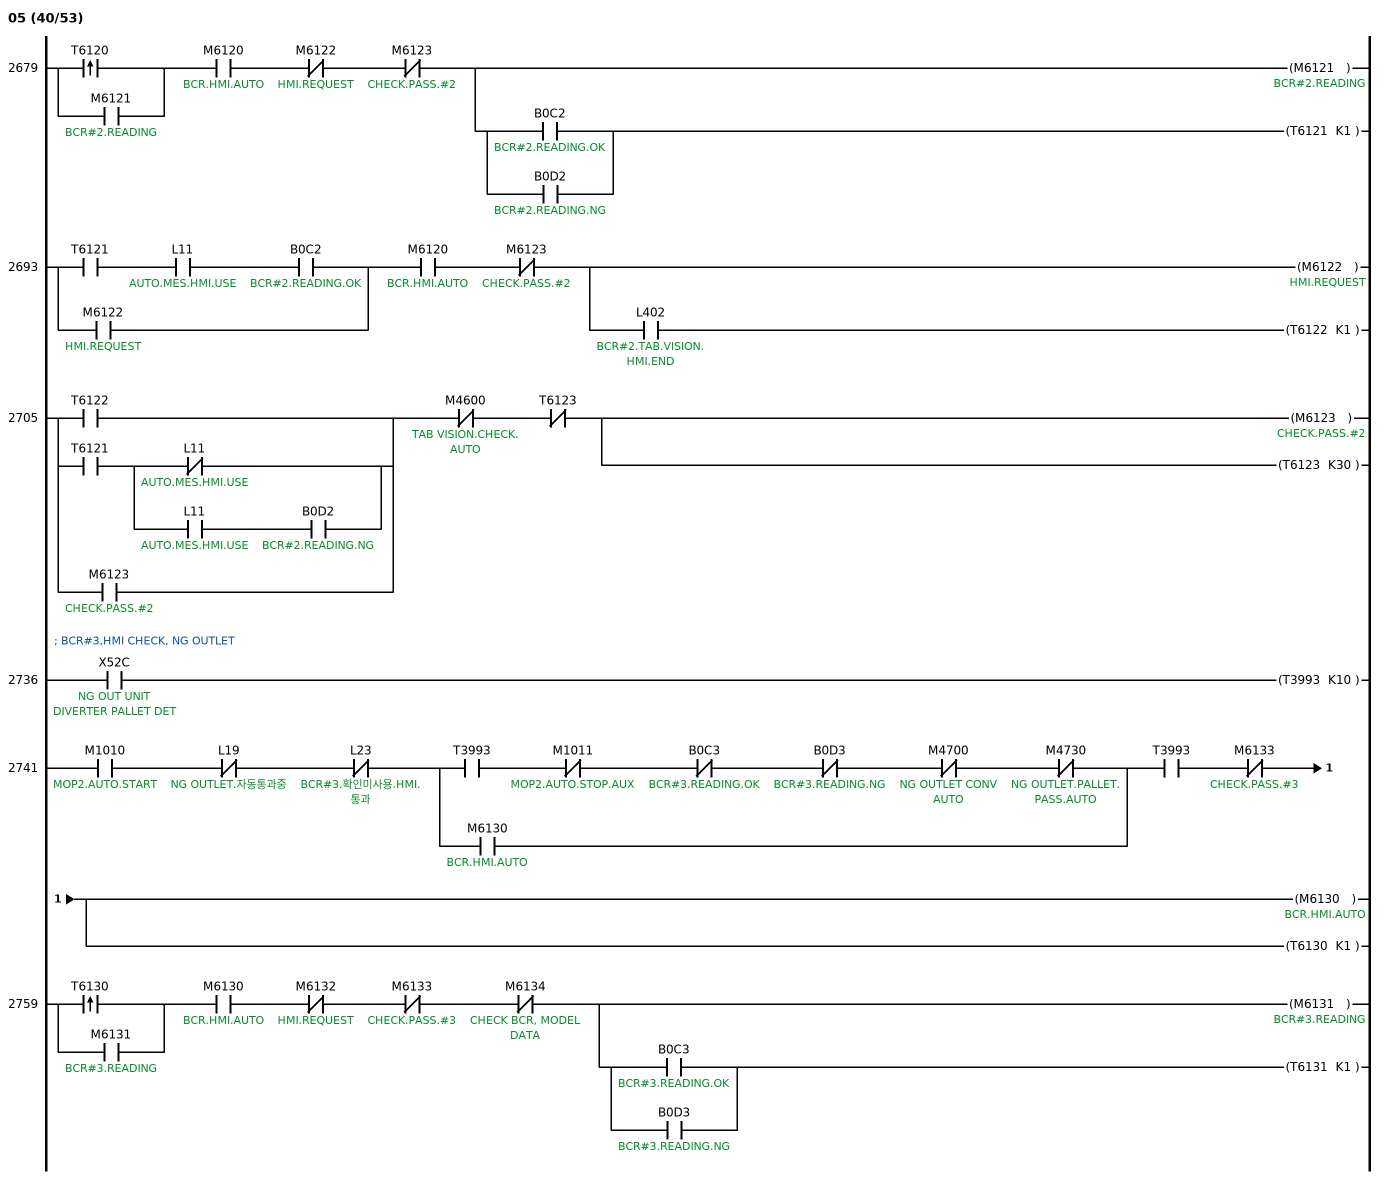
2679  LDP     T6120
      OR      M6121  ; BCR#2.READING
      AND     M6120  ; BCR.HMI.AUTO
      ANI     M6122  ; HMI.REQUEST
      ANI     M6123  ; CHECK.PASS.#2
      OUT     M6121  ; BCR#2.READING
      LD      B0C2  ; BCR#2.READING.OK
      OR      B0D2  ; BCR#2.READING.NG
      ANB
      OUT     T6121 K1
2693  LD      T6121
      AND     L11  ; AUTO.MES.HMI.USE
      AND     B0C2  ; BCR#2.READING.OK
      OR      M6122  ; HMI.REQUEST
      AND     M6120  ; BCR.HMI.AUTO
      ANI     M6123  ; CHECK.PASS.#2
      OUT     M6122  ; HMI.REQUEST
      AND     L402  ; BCR#2.TAB.VISION.HMI.END
      OUT     T6122 K1
2705  LD      T6122
      LD      T6121
      LDI     L11  ; AUTO.MES.HMI.USE
      LD      L11  ; AUTO.MES.HMI.USE
      AND     B0D2  ; BCR#2.READING.NG
      ORB
      ANB
      ORB
      OR      M6123  ; CHECK.PASS.#2
      ANI     M4600  ; TAB VISION.CHECK.AUTO
      ANI     T6123
      OUT     M6123  ; CHECK.PASS.#2
      OUT     T6123 K30
; BCR#3,HMI CHECK, NG OUTLET
2736  LD      X52C  ; NG OUT UNIT DIVERTER PALLET DET
      OUT     T3993 K10
2741  LD      M1010  ; MOP2.AUTO.START
      ANI     L19  ; NG OUTLET.자동통과중
      ANI     L23  ; BCR#3.확인미사용.HMI.통과
      LD      T3993
      ANI     M1011  ; MOP2.AUTO.STOP.AUX
      ANI     B0C3  ; BCR#3.READING.OK
      ANI     B0D3  ; BCR#3.READING.NG
      ANI     M4700  ; NG OUTLET CONV AUTO
      ANI     M4730  ; NG OUTLET.PALLET.PASS.AUTO
      OR      M6130  ; BCR.HMI.AUTO
      ANB
      AND     T3993
      ANI     M6133  ; CHECK.PASS.#3
      OUT     M6130  ; BCR.HMI.AUTO
      OUT     T6130 K1
2759  LDP     T6130
      OR      M6131  ; BCR#3.READING
      AND     M6130  ; BCR.HMI.AUTO
      ANI     M6132  ; HMI.REQUEST
      ANI     M6133  ; CHECK.PASS.#3
      ANI     M6134  ; CHECK BCR, MODEL DATA
      OUT     M6131  ; BCR#3.READING
      LD      B0C3  ; BCR#3.READING.OK
      OR      B0D3  ; BCR#3.READING.NG
      ANB
      OUT     T6131 K1
